// TIA Portal project "e215001v046" (V15)

(* hardware
DEVICE "Estación PC"  SIMATIC PC station
   slot 0: "Estación PC"  Rail  SIMATIC PC-Station  V1.0
      slot 125: "Stationmanager"  Station_Manager  V6.0.4
   slot 1: "IE general_1"  IE General  IE_CP  V8.2.0
   slot 2: "HMI_RT_1"  WinCC RT Advanced  6AV2 104-0xxxx-xxxx  15.0.0.0
      slot 33792: "Interfaz host"  Host interface
DEVICE "HMI_1"  KTP400 Basic mono PN
   slot 0: "HMI_1"  KTP400 Basic mono PN  6AV6 647-0AA11-3AX0  12.0.0.0
   slot 1: "HMI_RT_2"  KTP400 Basic mono PN  6AV6 647-0AA11-3AX0  12.0.0.0
   slot 5: "HMI_1.IE_CP_1"  PROFINET Interface  12.0.0.0
      slot 1: "Interfaz PROFINET_1"  PROFINET Interface
         slot 1: "Port_1"  Port
DEVICE "S7-1200 station_2"  S7-1200 Station
   slot 0: "Rack_0"  S7-1200 Rack  Rack  V1.0
   slot 1: "PLC_1"  CPU 1212C DC/DC/Rly  6ES7 212-1HE31-0XB0  V3.0
*)

// ===== PLC "PLC_1"  CPU 1212C DC/DC/Rly =====

VAR_GLOBAL   // PLC tag table "Tabla de variables estándar"
   "iSensIzqPla1" AT %I0.0 : Bool;
   "iSensMedPla1" AT %I0.1 : Bool;
   "iSensDerPla1" AT %I0.2 : Bool;
   "iMaqProdPla1" AT %I0.3 : Bool;
   "iSensIzqPla2" AT %I0.4 : Bool;
   "iSensMedPla2" AT %I0.5 : Bool;
   "iSensDerPla2" AT %I0.6 : Bool;
   "iMaqProdPla2" AT %I0.7 : Bool;
   "System_Byte" AT %MB1 : Byte;
   "FirstScan" AT %M1.0 : Bool;
   "DiagStatusUpdate" AT %M1.1 : Bool;
   "AlwaysTRUE" AT %M1.2 : Bool;
   "AlwaysFALSE" AT %M1.3 : Bool;
   "Clock_Byte" AT %MB0 : Byte;
   "Clock_10Hz" AT %M0.0 : Bool;
   "Clock_5Hz" AT %M0.1 : Bool;
   "Clock_2.5Hz" AT %M0.2 : Bool;
   "Clock_2Hz" AT %M0.3 : Bool;
   "Clock_1.25Hz" AT %M0.4 : Bool;
   "Clock_1Hz" AT %M0.5 : Bool;
   "Clock_0.625Hz" AT %M0.6 : Bool;
   "Clock_0.5Hz" AT %M0.7 : Bool;
   "fClock_10Hz" AT %M2.0 : Bool;
   "xClock_10Hz" AT %M2.1 : Bool;
   "Plan1EnProd" AT %M2.2 : Bool;
   "Plan1Ok" AT %M2.3 : Bool;
   "Tag_1" AT %M10.0 : Bool;
   "Tag_2" AT %M10.1 : Bool;
   "Tag_3" AT %M10.2 : Bool;
   "Tag_4" AT %M10.3 : Bool;
   "Tag_5" AT %M11.0 : Bool;
   "Tag_6" AT %M11.1 : Bool;
   "Tag_7" AT %M11.2 : Bool;
   "Tag_8" AT %M11.3 : Bool;
   "Flc_Asc_Planch1_10Hz" AT %M501.0 : Bool;
   "Flc_Asc_Planch2_10Hz" AT %M501.1 : Bool;
   "Rec_Alarm" AT %M5.0 : Bool;
   "Osc_5mins" AT %M100.0 : Bool;
   "Palabra Distr" AT %MB101 : Byte;
   "PFlc_SnsMed" AT %M100.1 : Bool;
   "Act_Simu" AT %M1000.0 : Bool;
   "HMI_Supervisor_Actual" AT %M50.0 : Bool;
   "periodoPlanchas" AT %MD110 : DInt;
   "promedioAvanceReal" AT %MD114 : Real;
   "contPromAvReal" AT %MD118 : DInt;
   "tmp_avanceReal_1" AT %MD122 : Real;
   "doProm" AT %M50.1 : Bool;
   "doProm_calculo" AT %M50.2 : Bool;
   "promDone" AT %M50.3 : Bool;
   "Tag_9" AT %M50.4 : Bool;
END_VAR

VAR_GLOBAL   // PLC tag table "DIDO"
   "fSup1" AT %M2.4 : Bool;
   "xsup1" AT %M2.5 : Bool;
   "fSup2" AT %M2.6 : Bool;
   "xsup2" AT %M2.7 : Bool;
   "fSup3" AT %M3.0 : Bool;
   "xsup3" AT %M3.1 : Bool;
   "fSup4" AT %M3.2 : Bool;
   "xsup4" AT %M3.3 : Bool;
   "Cada15M" AT %M3.4 : Bool;
   "fCada15M" AT %M3.5 : Bool;
   "xCada15M" AT %M3.6 : Bool;
   "Supervision" AT %M3.7 : Bool;
   "Plan2EnProd" AT %M4.3 : Bool;
   "Plan2Ok" AT %M4.7 : Bool;
END_VAR

DATA_BLOCK "Planchadora1"   // DB1
{ S7_Optimized_Access := 'TRUE' }
VERSION : 0.1
   VAR RETAIN
      Operadores : Array[1..10] of Struct
         Tiempo : DInt;
         Produccion : DInt;
         Productividad : DInt;
         Sensor : DInt;
         Rendimiento : DInt;
         RendPesado : DInt;
         Estado : Bool;
         Diadelasemana : Array[1..7] of Struct
            Entrda : Time_Of_Day;
            Salida : Time_Of_Day;
         END_STRUCT;
      END_STRUCT;
      Supervisores : Array[1..4] of Struct
         Tiempo : DInt;
         Produccion : DInt;
         Productividad : DInt;
         Sensor : DInt;
         Rendimiento : DInt;
         RendPesado : DInt;
         Estado : Bool;
         Diadelasemana : Array[1..7] of Struct
            Entrada : Time_Of_Day;
            Salida : Time_Of_Day;
            CantOp : Int;
         END_STRUCT;
      END_STRUCT;
      FechaHoraPLC : DTL := DTL#2020-03-12-10:25:17.055662;
      ProductividadTotal : DInt := 861_100_900;
      Productividad : DInt := 0;
      Productividad_100 : Real := 0.0;
      TiempoTotal : DInt := 978_227_090;
      Tiempo : DInt := 511710;
      RendimientoTotal : DInt := 246_159_997;
      Rendimiento : DInt := 0;
   END_VAR
   VAR
      DifRendimiento : DInt := 0;
   END_VAR
   VAR RETAIN
      Rendimiento_100 : Real := 39.44824;
      RendPesado : DInt := 244_381_165;
      RendPesado_100 : Real := 970325.3;
      Productividad_Verde : Real := 0.0;
      Productividad_Amarillo : Real := 0.0;
      Productividad_Rojo : Real := 0.0;
      Rendimiento_Verde : Real := 0.0;
      Rendimiento_Amarillo : Real := 0.0;
      Rendimiento_Rojo : Real := 0.0;
      Peso_Sensor : Int := 0;
      Peso_SensorIZq : Int := 0;
      Peso_SensorDer : Int := 0;
      Peso_SensorMed : Int := 0;
      TiempoCada15 : DInt := 0;
      ProductividadCada15 : DInt := 0;
      RendimientoCada15 : DInt := 0;
      TiempoCada15Ant : DInt := 978_165_380;
      ProductividadCada15Ant : DInt := 861_100_900;
      RendimientoCada15Ant : DInt := 246_159_997;
      EstadoSsIzq : Byte := 16#00;
      EstadoSsDer : Byte := 16#00;
      EstadoSSMed : Byte := 16#00;
   END_VAR
   VAR
      SumaOperario : Int := 1;
   END_VAR
   VAR RETAIN
      FactorCorrRend : Real := 2.0;
   END_VAR
BEGIN
   Operadores[1].Tiempo := 0;
   Operadores[1].Produccion := 0;
   Operadores[1].Productividad := 0;
   Operadores[1].Sensor := 0;
   Operadores[1].Rendimiento := 0;
   Operadores[1].RendPesado := 0;
   Operadores[1].Estado := FALSE;
   Operadores[1].Diadelasemana[1].Entrda := TOD#00:00:00;
   Operadores[1].Diadelasemana[1].Salida := TOD#00:00:00;
   Operadores[1].Diadelasemana[2].Entrda := TOD#00:00:00;
   Operadores[1].Diadelasemana[2].Salida := TOD#00:00:00;
   Operadores[1].Diadelasemana[3].Entrda := TOD#00:00:00;
   Operadores[1].Diadelasemana[3].Salida := TOD#00:00:00;
   Operadores[1].Diadelasemana[4].Entrda := TOD#00:00:00;
   Operadores[1].Diadelasemana[4].Salida := TOD#00:00:00;
   Operadores[1].Diadelasemana[5].Entrda := TOD#00:00:00;
   Operadores[1].Diadelasemana[5].Salida := TOD#00:00:00;
   Operadores[1].Diadelasemana[6].Entrda := TOD#00:00:00;
   Operadores[1].Diadelasemana[6].Salida := TOD#00:00:00;
   Operadores[1].Diadelasemana[7].Entrda := TOD#00:00:00;
   Operadores[1].Diadelasemana[7].Salida := TOD#00:00:00;
   Operadores[2].Tiempo := 0;
   Operadores[2].Produccion := 0;
   Operadores[2].Productividad := 0;
   Operadores[2].Sensor := 0;
   Operadores[2].Rendimiento := 0;
   Operadores[2].RendPesado := 0;
   Operadores[2].Estado := FALSE;
   Operadores[2].Diadelasemana[1].Entrda := TOD#00:00:00;
   Operadores[2].Diadelasemana[1].Salida := TOD#00:00:00;
   Operadores[2].Diadelasemana[2].Entrda := TOD#00:00:00;
   Operadores[2].Diadelasemana[2].Salida := TOD#00:00:00;
   Operadores[2].Diadelasemana[3].Entrda := TOD#00:00:00;
   Operadores[2].Diadelasemana[3].Salida := TOD#00:00:00;
   Operadores[2].Diadelasemana[4].Entrda := TOD#00:00:00;
   Operadores[2].Diadelasemana[4].Salida := TOD#00:00:00;
   Operadores[2].Diadelasemana[5].Entrda := TOD#00:00:00;
   Operadores[2].Diadelasemana[5].Salida := TOD#00:00:00;
   Operadores[2].Diadelasemana[6].Entrda := TOD#00:00:00;
   Operadores[2].Diadelasemana[6].Salida := TOD#00:00:00;
   Operadores[2].Diadelasemana[7].Entrda := TOD#00:00:00;
   Operadores[2].Diadelasemana[7].Salida := TOD#00:00:00;
   Operadores[3].Tiempo := 0;
   Operadores[3].Produccion := 0;
   Operadores[3].Productividad := 0;
   Operadores[3].Sensor := 0;
   Operadores[3].Rendimiento := 0;
   Operadores[3].RendPesado := 0;
   Operadores[3].Estado := FALSE;
   Operadores[3].Diadelasemana[1].Entrda := TOD#00:00:00;
   Operadores[3].Diadelasemana[1].Salida := TOD#00:00:00;
   Operadores[3].Diadelasemana[2].Entrda := TOD#00:00:00;
   Operadores[3].Diadelasemana[2].Salida := TOD#00:00:00;
   Operadores[3].Diadelasemana[3].Entrda := TOD#00:00:00;
   Operadores[3].Diadelasemana[3].Salida := TOD#00:00:00;
   Operadores[3].Diadelasemana[4].Entrda := TOD#00:00:00;
   Operadores[3].Diadelasemana[4].Salida := TOD#00:00:00;
   Operadores[3].Diadelasemana[5].Entrda := TOD#00:00:00;
   Operadores[3].Diadelasemana[5].Salida := TOD#00:00:00;
   Operadores[3].Diadelasemana[6].Entrda := TOD#00:00:00;
   Operadores[3].Diadelasemana[6].Salida := TOD#00:00:00;
   Operadores[3].Diadelasemana[7].Entrda := TOD#00:00:00;
   Operadores[3].Diadelasemana[7].Salida := TOD#00:00:00;
   Operadores[4].Tiempo := 55366140;
   Operadores[4].Produccion := 49275400;
   Operadores[4].Productividad := 0;
   Operadores[4].Sensor := 0;
   Operadores[4].Rendimiento := 12680067;
   Operadores[4].RendPesado := 12605331;
   Operadores[4].Estado := FALSE;
   Operadores[4].Diadelasemana[1].Entrda := TOD#00:00:00;
   Operadores[4].Diadelasemana[1].Salida := TOD#00:00:00;
   Operadores[4].Diadelasemana[2].Entrda := TOD#00:00:00;
   Operadores[4].Diadelasemana[2].Salida := TOD#00:00:00;
   Operadores[4].Diadelasemana[3].Entrda := TOD#00:00:00;
   Operadores[4].Diadelasemana[3].Salida := TOD#00:00:00;
   Operadores[4].Diadelasemana[4].Entrda := TOD#00:00:00;
   Operadores[4].Diadelasemana[4].Salida := TOD#00:00:00;
   Operadores[4].Diadelasemana[5].Entrda := TOD#00:00:00;
   Operadores[4].Diadelasemana[5].Salida := TOD#00:00:00;
   Operadores[4].Diadelasemana[6].Entrda := TOD#00:00:00;
   Operadores[4].Diadelasemana[6].Salida := TOD#00:00:00;
   Operadores[4].Diadelasemana[7].Entrda := TOD#00:00:00;
   Operadores[4].Diadelasemana[7].Salida := TOD#00:00:00;
   Operadores[5].Tiempo := 976_354_630;
   Operadores[5].Produccion := 859_251_080;
   Operadores[5].Productividad := 0;
   Operadores[5].Sensor := 0;
   Operadores[5].Rendimiento := 245_655_295;
   Operadores[5].RendPesado := 243_132_090;
   Operadores[5].Estado := TRUE;
   Operadores[5].Diadelasemana[1].Entrda := TOD#00:00:00;
   Operadores[5].Diadelasemana[1].Salida := TOD#00:00:00;
   Operadores[5].Diadelasemana[2].Entrda := TOD#00:00:00;
   Operadores[5].Diadelasemana[2].Salida := TOD#00:00:00;
   Operadores[5].Diadelasemana[3].Entrda := TOD#00:00:00;
   Operadores[5].Diadelasemana[3].Salida := TOD#00:00:00;
   Operadores[5].Diadelasemana[4].Entrda := TOD#00:00:00;
   Operadores[5].Diadelasemana[4].Salida := TOD#00:00:00;
   Operadores[5].Diadelasemana[5].Entrda := TOD#00:00:00;
   Operadores[5].Diadelasemana[5].Salida := TOD#00:00:00;
   Operadores[5].Diadelasemana[6].Entrda := TOD#00:00:00;
   Operadores[5].Diadelasemana[6].Salida := TOD#00:00:00;
   Operadores[5].Diadelasemana[7].Entrda := TOD#00:00:00;
   Operadores[5].Diadelasemana[7].Salida := TOD#00:00:00;
   Operadores[6].Tiempo := 0;
   Operadores[6].Produccion := 0;
   Operadores[6].Productividad := 0;
   Operadores[6].Sensor := 0;
   Operadores[6].Rendimiento := 0;
   Operadores[6].RendPesado := 0;
   Operadores[6].Estado := FALSE;
   Operadores[6].Diadelasemana[1].Entrda := TOD#00:00:00;
   Operadores[6].Diadelasemana[1].Salida := TOD#00:00:00;
   Operadores[6].Diadelasemana[2].Entrda := TOD#00:00:00;
   Operadores[6].Diadelasemana[2].Salida := TOD#00:00:00;
   Operadores[6].Diadelasemana[3].Entrda := TOD#00:00:00;
   Operadores[6].Diadelasemana[3].Salida := TOD#00:00:00;
   Operadores[6].Diadelasemana[4].Entrda := TOD#00:00:00;
   Operadores[6].Diadelasemana[4].Salida := TOD#00:00:00;
   Operadores[6].Diadelasemana[5].Entrda := TOD#00:00:00;
   Operadores[6].Diadelasemana[5].Salida := TOD#00:00:00;
   Operadores[6].Diadelasemana[6].Entrda := TOD#00:00:00;
   Operadores[6].Diadelasemana[6].Salida := TOD#00:00:00;
   Operadores[6].Diadelasemana[7].Entrda := TOD#00:00:00;
   Operadores[6].Diadelasemana[7].Salida := TOD#00:00:00;
   Operadores[7].Tiempo := 0;
   Operadores[7].Produccion := 0;
   Operadores[7].Productividad := 0;
   Operadores[7].Sensor := 0;
   Operadores[7].Rendimiento := 0;
   Operadores[7].RendPesado := 0;
   Operadores[7].Estado := FALSE;
   Operadores[7].Diadelasemana[1].Entrda := TOD#00:00:00;
   Operadores[7].Diadelasemana[1].Salida := TOD#00:00:00;
   Operadores[7].Diadelasemana[2].Entrda := TOD#00:00:00;
   Operadores[7].Diadelasemana[2].Salida := TOD#00:00:00;
   Operadores[7].Diadelasemana[3].Entrda := TOD#00:00:00;
   Operadores[7].Diadelasemana[3].Salida := TOD#00:00:00;
   Operadores[7].Diadelasemana[4].Entrda := TOD#00:00:00;
   Operadores[7].Diadelasemana[4].Salida := TOD#00:00:00;
   Operadores[7].Diadelasemana[5].Entrda := TOD#00:00:00;
   Operadores[7].Diadelasemana[5].Salida := TOD#00:00:00;
   Operadores[7].Diadelasemana[6].Entrda := TOD#00:00:00;
   Operadores[7].Diadelasemana[6].Salida := TOD#00:00:00;
   Operadores[7].Diadelasemana[7].Entrda := TOD#00:00:00;
   Operadores[7].Diadelasemana[7].Salida := TOD#00:00:00;
   Operadores[8].Tiempo := 0;
   Operadores[8].Produccion := 0;
   Operadores[8].Productividad := 0;
   Operadores[8].Sensor := 0;
   Operadores[8].Rendimiento := 0;
   Operadores[8].RendPesado := 0;
   Operadores[8].Estado := FALSE;
   Operadores[8].Diadelasemana[1].Entrda := TOD#00:00:00;
   Operadores[8].Diadelasemana[1].Salida := TOD#00:00:00;
   Operadores[8].Diadelasemana[2].Entrda := TOD#00:00:00;
   Operadores[8].Diadelasemana[2].Salida := TOD#00:00:00;
   Operadores[8].Diadelasemana[3].Entrda := TOD#00:00:00;
   Operadores[8].Diadelasemana[3].Salida := TOD#00:00:00;
   Operadores[8].Diadelasemana[4].Entrda := TOD#00:00:00;
   Operadores[8].Diadelasemana[4].Salida := TOD#00:00:00;
   Operadores[8].Diadelasemana[5].Entrda := TOD#00:00:00;
   Operadores[8].Diadelasemana[5].Salida := TOD#00:00:00;
   Operadores[8].Diadelasemana[6].Entrda := TOD#00:00:00;
   Operadores[8].Diadelasemana[6].Salida := TOD#00:00:00;
   Operadores[8].Diadelasemana[7].Entrda := TOD#00:00:00;
   Operadores[8].Diadelasemana[7].Salida := TOD#00:00:00;
   Operadores[9].Tiempo := 0;
   Operadores[9].Produccion := 0;
   Operadores[9].Productividad := 0;
   Operadores[9].Sensor := 0;
   Operadores[9].Rendimiento := 0;
   Operadores[9].RendPesado := 0;
   Operadores[9].Estado := FALSE;
   Operadores[9].Diadelasemana[1].Entrda := TOD#00:00:00;
   Operadores[9].Diadelasemana[1].Salida := TOD#00:00:00;
   Operadores[9].Diadelasemana[2].Entrda := TOD#00:00:00;
   Operadores[9].Diadelasemana[2].Salida := TOD#00:00:00;
   Operadores[9].Diadelasemana[3].Entrda := TOD#00:00:00;
   Operadores[9].Diadelasemana[3].Salida := TOD#00:00:00;
   Operadores[9].Diadelasemana[4].Entrda := TOD#00:00:00;
   Operadores[9].Diadelasemana[4].Salida := TOD#00:00:00;
   Operadores[9].Diadelasemana[5].Entrda := TOD#00:00:00;
   Operadores[9].Diadelasemana[5].Salida := TOD#00:00:00;
   Operadores[9].Diadelasemana[6].Entrda := TOD#00:00:00;
   Operadores[9].Diadelasemana[6].Salida := TOD#00:00:00;
   Operadores[9].Diadelasemana[7].Entrda := TOD#00:00:00;
   Operadores[9].Diadelasemana[7].Salida := TOD#00:00:00;
   Operadores[10].Tiempo := 2860;
   Operadores[10].Produccion := 2860;
   Operadores[10].Productividad := 0;
   Operadores[10].Sensor := 0;
   Operadores[10].Rendimiento := 281;
   Operadores[10].RendPesado := 0;
   Operadores[10].Estado := FALSE;
   Operadores[10].Diadelasemana[1].Entrda := TOD#00:00:00;
   Operadores[10].Diadelasemana[1].Salida := TOD#00:00:00;
   Operadores[10].Diadelasemana[2].Entrda := TOD#00:00:00;
   Operadores[10].Diadelasemana[2].Salida := TOD#00:00:00;
   Operadores[10].Diadelasemana[3].Entrda := TOD#00:00:00;
   Operadores[10].Diadelasemana[3].Salida := TOD#00:00:00;
   Operadores[10].Diadelasemana[4].Entrda := TOD#00:00:00;
   Operadores[10].Diadelasemana[4].Salida := TOD#00:00:00;
   Operadores[10].Diadelasemana[5].Entrda := TOD#00:00:00;
   Operadores[10].Diadelasemana[5].Salida := TOD#00:00:00;
   Operadores[10].Diadelasemana[6].Entrda := TOD#00:00:00;
   Operadores[10].Diadelasemana[6].Salida := TOD#00:00:00;
   Operadores[10].Diadelasemana[7].Entrda := TOD#00:00:00;
   Operadores[10].Diadelasemana[7].Salida := TOD#00:00:00;
   Supervisores[1].Tiempo := 253_394_970;
   Supervisores[1].Produccion := 229_902_840;
   Supervisores[1].Productividad := 0;
   Supervisores[1].Sensor := 0;
   Supervisores[1].Rendimiento := 65119768;
   Supervisores[1].RendPesado := 2880135;
   Supervisores[1].Estado := FALSE;
   Supervisores[1].Diadelasemana[1].Entrada := TOD#00:00:00;
   Supervisores[1].Diadelasemana[1].Salida := TOD#00:00:00;
   Supervisores[1].Diadelasemana[1].CantOp := 1;
   Supervisores[1].Diadelasemana[2].Entrada := TOD#06:00:00;
   Supervisores[1].Diadelasemana[2].Salida := TOD#09:00:00;
   Supervisores[1].Diadelasemana[2].CantOp := 1;
   Supervisores[1].Diadelasemana[3].Entrada := TOD#06:00:00;
   Supervisores[1].Diadelasemana[3].Salida := TOD#09:00:00;
   Supervisores[1].Diadelasemana[3].CantOp := 1;
   Supervisores[1].Diadelasemana[4].Entrada := TOD#06:00:00;
   Supervisores[1].Diadelasemana[4].Salida := TOD#09:00:00;
   Supervisores[1].Diadelasemana[4].CantOp := 1;
   Supervisores[1].Diadelasemana[5].Entrada := TOD#06:00:00;
   Supervisores[1].Diadelasemana[5].Salida := TOD#09:00:00;
   Supervisores[1].Diadelasemana[5].CantOp := 1;
   Supervisores[1].Diadelasemana[6].Entrada := TOD#06:00:00;
   Supervisores[1].Diadelasemana[6].Salida := TOD#09:00:00;
   Supervisores[1].Diadelasemana[6].CantOp := 1;
   Supervisores[1].Diadelasemana[7].Entrada := TOD#06:00:00;
   Supervisores[1].Diadelasemana[7].Salida := TOD#14:00:00;
   Supervisores[1].Diadelasemana[7].CantOp := 1;
   Supervisores[2].Tiempo := 427_440_520;
   Supervisores[2].Produccion := 385_662_930;
   Supervisores[2].Productividad := 0;
   Supervisores[2].Sensor := 0;
   Supervisores[2].Rendimiento := 113_827_501;
   Supervisores[2].RendPesado := 3250056;
   Supervisores[2].Estado := TRUE;
   Supervisores[2].Diadelasemana[1].Entrada := TOD#00:00:00;
   Supervisores[2].Diadelasemana[1].Salida := TOD#00:00:00;
   Supervisores[2].Diadelasemana[1].CantOp := 1;
   Supervisores[2].Diadelasemana[2].Entrada := TOD#09:00:00;
   Supervisores[2].Diadelasemana[2].Salida := TOD#17:00:00;
   Supervisores[2].Diadelasemana[2].CantOp := 1;
   Supervisores[2].Diadelasemana[3].Entrada := TOD#09:00:00;
   Supervisores[2].Diadelasemana[3].Salida := TOD#17:00:00;
   Supervisores[2].Diadelasemana[3].CantOp := 1;
   Supervisores[2].Diadelasemana[4].Entrada := TOD#09:00:00;
   Supervisores[2].Diadelasemana[4].Salida := TOD#17:00:00;
   Supervisores[2].Diadelasemana[4].CantOp := 1;
   Supervisores[2].Diadelasemana[5].Entrada := TOD#09:00:00;
   Supervisores[2].Diadelasemana[5].Salida := TOD#17:00:00;
   Supervisores[2].Diadelasemana[5].CantOp := 1;
   Supervisores[2].Diadelasemana[6].Entrada := TOD#09:00:00;
   Supervisores[2].Diadelasemana[6].Salida := TOD#17:00:00;
   Supervisores[2].Diadelasemana[6].CantOp := 1;
   Supervisores[2].Diadelasemana[7].Entrada := TOD#14:00:00;
   Supervisores[2].Diadelasemana[7].Salida := TOD#22:00:00;
   Supervisores[2].Diadelasemana[7].CantOp := 1;
   Supervisores[3].Tiempo := 297_391_250;
   Supervisores[3].Produccion := 245_534_940;
   Supervisores[3].Productividad := 0;
   Supervisores[3].Sensor := 0;
   Supervisores[3].Rendimiento := 67212726;
   Supervisores[3].RendPesado := 2469772;
   Supervisores[3].Estado := FALSE;
   Supervisores[3].Diadelasemana[1].Entrada := TOD#06:00:00;
   Supervisores[3].Diadelasemana[1].Salida := TOD#14:00:00;
   Supervisores[3].Diadelasemana[1].CantOp := 1;
   Supervisores[3].Diadelasemana[2].Entrada := TOD#17:00:00;
   Supervisores[3].Diadelasemana[2].Salida := TOD#22:00:00;
   Supervisores[3].Diadelasemana[2].CantOp := 1;
   Supervisores[3].Diadelasemana[3].Entrada := TOD#17:00:00;
   Supervisores[3].Diadelasemana[3].Salida := TOD#22:00:00;
   Supervisores[3].Diadelasemana[3].CantOp := 1;
   Supervisores[3].Diadelasemana[4].Entrada := TOD#17:00:00;
   Supervisores[3].Diadelasemana[4].Salida := TOD#22:00:00;
   Supervisores[3].Diadelasemana[4].CantOp := 1;
   Supervisores[3].Diadelasemana[5].Entrada := TOD#17:00:00;
   Supervisores[3].Diadelasemana[5].Salida := TOD#22:00:00;
   Supervisores[3].Diadelasemana[5].CantOp := 1;
   Supervisores[3].Diadelasemana[6].Entrada := TOD#17:00:00;
   Supervisores[3].Diadelasemana[6].Salida := TOD#22:00:00;
   Supervisores[3].Diadelasemana[6].CantOp := 1;
   Supervisores[3].Diadelasemana[7].Entrada := TOD#00:00:00;
   Supervisores[3].Diadelasemana[7].Salida := TOD#00:00:00;
   Supervisores[3].Diadelasemana[7].CantOp := 1;
   Supervisores[4].Tiempo := 0;
   Supervisores[4].Produccion := 0;
   Supervisores[4].Productividad := 0;
   Supervisores[4].Sensor := 0;
   Supervisores[4].Rendimiento := 0;
   Supervisores[4].RendPesado := 0;
   Supervisores[4].Estado := FALSE;
   Supervisores[4].Diadelasemana[1].Entrada := TOD#00:00:00;
   Supervisores[4].Diadelasemana[1].Salida := TOD#00:00:00;
   Supervisores[4].Diadelasemana[1].CantOp := 1;
   Supervisores[4].Diadelasemana[2].Entrada := TOD#00:00:00;
   Supervisores[4].Diadelasemana[2].Salida := TOD#00:00:00;
   Supervisores[4].Diadelasemana[2].CantOp := 1;
   Supervisores[4].Diadelasemana[3].Entrada := TOD#00:00:00;
   Supervisores[4].Diadelasemana[3].Salida := TOD#00:00:00;
   Supervisores[4].Diadelasemana[3].CantOp := 1;
   Supervisores[4].Diadelasemana[4].Entrada := TOD#00:00:00;
   Supervisores[4].Diadelasemana[4].Salida := TOD#00:00:00;
   Supervisores[4].Diadelasemana[4].CantOp := 1;
   Supervisores[4].Diadelasemana[5].Entrada := TOD#00:00:00;
   Supervisores[4].Diadelasemana[5].Salida := TOD#00:00:00;
   Supervisores[4].Diadelasemana[5].CantOp := 1;
   Supervisores[4].Diadelasemana[6].Entrada := TOD#00:00:00;
   Supervisores[4].Diadelasemana[6].Salida := TOD#00:00:00;
   Supervisores[4].Diadelasemana[6].CantOp := 1;
   Supervisores[4].Diadelasemana[7].Entrada := TOD#00:00:00;
   Supervisores[4].Diadelasemana[7].Salida := TOD#00:00:00;
   Supervisores[4].Diadelasemana[7].CantOp := 1;
END_DATA_BLOCK

DATA_BLOCK "Planchadora2"   // DB5
{ S7_Optimized_Access := 'TRUE' }
VERSION : 0.1
   VAR RETAIN
      Operadores : Array[1..10] of Struct
         Tiempo : DInt;
         Produccion : DInt;
         Productividad : DInt;
         Sensor : DInt;
         Rendimiento : DInt;
         RendPesado : DInt;
         Estado : Bool;
         Diadelasemana : Array[1..7] of Struct
            Entrda : Time_Of_Day;
            Salida : Time_Of_Day;
         END_STRUCT;
      END_STRUCT;
      Supervisores : Array[1..4] of Struct
         Tiempo : DInt;
         Produccion : DInt;
         Productividad : DInt;
         Sensor : DInt;
         Rendimiento : DInt;
         RendPesado : DInt;
         Estado : Bool;
         Diadelasemana : Array[1..7] of Struct
            Entrada : Time_Of_Day;
            Salida : Time_Of_Day;
            CantOp : Int;
         END_STRUCT;
      END_STRUCT;
      FechaHoraPLC : DTL;
      ProductividadTotal : DInt;
      Productividad : DInt;
      Productividad_100 : Real;
      TiempoTotal : DInt;
      Tiempo : DInt;
      RendimientoTotal : DInt;
      Rendimiento : DInt;
   END_VAR
   VAR
      DifRendimiento : DInt;
   END_VAR
   VAR RETAIN
      Rendimiento_100 : Real;
      RendPesado : DInt;
      RendPesado_100 : Real;
      Productividad_Verde : Real;
      Productividad_Amarillo : Real;
      Productividad_Rojo : Real;
      Rendimiento_Verde : Real;
      Rendimiento_Amarillo : Real;
      Rendimiento_Rojo : Real;
      Peso_Sensor : Int;
      Peso_SensorIZq : Int;
      Peso_SensorDer : Int;
      Peso_SensorMed : Int;
      TiempoCada15 : DInt;
      ProductividadCada15 : DInt;
      RendimientoCada15 : DInt;
      TiempoCada15Ant : DInt;
      ProductividadCada15Ant : DInt;
      RendimientoCada15Ant : DInt;
      EstadoSsIzq : Byte;
      EstadoSsDer : Byte;
      EstadoSSMed : Byte;
      FechayhoraS : String := '1970-01-00-00-00:00:00';
   END_VAR
   VAR
      SumaOperario : Int;
   END_VAR
   VAR RETAIN
      FactorCorrRend : Real := 3.0;
   END_VAR
BEGIN
END_DATA_BLOCK

DATA_BLOCK "Alarmas"   // DB9
{ S7_Optimized_Access := 'FALSE' }
VERSION : 0.1
   VAR
      "PL1-Fall-SnsIzq" : Bool;
      "PL1-Fall-SnsMed" : Bool;
      "PL1-Fall-SnsDer" : Bool;
      "PL2-Fall-SnsIzq" : Bool;
      "PL2-Fall-SnsMed" : Bool;
      "PL2-Fall-SnsDer" : Bool;
      Gen_6 : Bool;
      Gen_7 : Bool;
      Gen_8 : Bool;
      Gen_9 : Bool;
      Gen_10 : Bool;
      Gen_11 : Bool;
      Gen_12 : Bool;
      Gen_13 : Bool;
      Gen_14 : Bool;
      Gen_15 : Bool;
      Gen_16 : Bool;
      Gen_17 : Bool;
      Gen_18 : Bool;
      Gen_19 : Bool;
      Gen_20 : Bool;
      Gen_21 : Bool;
      Gen_22 : Bool;
      Gen_23 : Bool;
      Gen_24 : Bool;
      Gen_25 : Bool;
      Gen_26 : Bool;
      Gen_27 : Bool;
      Gen_28 : Bool;
      Gen_29 : Bool;
      Gen_30 : Bool;
      Gen_31 : Bool;
   END_VAR
BEGIN
END_DATA_BLOCK

DATA_BLOCK "00_ValoresdeReferencia"   // DB11
{ S7_Optimized_Access := 'TRUE' }
VERSION : 0.1
   VAR RETAIN
      pl1_ProdTotal_Ant : DInt;
      pl1_RendTotal_Ant : DInt;
      pl2_ProdTotal_Ant : DInt;
      pl2_RendTotal_Ant : DInt;
   END_VAR
BEGIN
END_DATA_BLOCK

DATA_BLOCK "TratCentecimasSeg"   // DB13
{ S7_Optimized_Access := 'TRUE' }
VERSION : 0.1
   VAR
      Pl1_Cen_SnsIzq : Int;
      Pl1_Cen_SnsMed : Int;
      Pl1_Cen_SnsDer : Int;
      Pl2_Cen_SnsIzq : Int;
      Pl2_Cen_SnsMed : Int;
      Pl2_Cen_SnsDer : Int;
   END_VAR
BEGIN
END_DATA_BLOCK

DATA_BLOCK "Indices"   // DB14
{ S7_Optimized_Access := 'TRUE' }
VERSION : 0.1
   VAR RETAIN
      horasTurno : Time_Of_Day;
      objetivo_100 : Real;
      objetivo : Time_Of_Day;
      avance : Time_Of_Day;
      avance_100 : Real;
      avance_real : Time_Of_Day;
      avance_real_100 : Real;
   END_VAR
BEGIN
END_DATA_BLOCK

// folder: System blocks/Program resources

DATA_BLOCK "tFaSsIzqPl1"   // DB2
{ S7_Optimized_Access := 'TRUE' }
AUTHOR : Simatic
FAMILY : IEC
NAME : IEC_TMR
VERSION : 1.0
// stored: InstanceOfName IEC_TIMER
"IEC_TIMER"
BEGIN
END_DATA_BLOCK

DATA_BLOCK "tFaSsMedPl1"   // DB3
{ S7_Optimized_Access := 'TRUE' }
AUTHOR : Simatic
FAMILY : IEC
NAME : IEC_TMR
VERSION : 1.0
// stored: InstanceOfName IEC_TIMER
"IEC_TIMER"
BEGIN
END_DATA_BLOCK

DATA_BLOCK "tFaSsDerPl1"   // DB4
{ S7_Optimized_Access := 'TRUE' }
AUTHOR : Simatic
FAMILY : IEC
NAME : IEC_TMR
VERSION : 1.0
// stored: InstanceOfName IEC_TIMER
"IEC_TIMER"
BEGIN
END_DATA_BLOCK

DATA_BLOCK "tFaSsIzqPl2"   // DB6
{ S7_Optimized_Access := 'TRUE' }
AUTHOR : Simatic
FAMILY : IEC
NAME : IEC_TMR
VERSION : 1.0
// stored: InstanceOfName IEC_TIMER
"IEC_TIMER"
BEGIN
END_DATA_BLOCK

DATA_BLOCK "tFaSsMedPl2"   // DB7
{ S7_Optimized_Access := 'TRUE' }
AUTHOR : Simatic
FAMILY : IEC
NAME : IEC_TMR
VERSION : 1.0
// stored: InstanceOfName IEC_TIMER
"IEC_TIMER"
BEGIN
END_DATA_BLOCK

DATA_BLOCK "tFaSsDerPl2"   // DB8
{ S7_Optimized_Access := 'TRUE' }
AUTHOR : Simatic
FAMILY : IEC
NAME : IEC_TMR
VERSION : 1.0
// stored: InstanceOfName IEC_TIMER
"IEC_TIMER"
BEGIN
END_DATA_BLOCK

DATA_BLOCK "IEC_Timer_0_DB"   // DB10
{ S7_Optimized_Access := 'TRUE' }
AUTHOR : Simatic
FAMILY : IEC
NAME : IEC_TMR
VERSION : 1.0
// stored: InstanceOfName IEC_TIMER
"IEC_TIMER"
BEGIN
END_DATA_BLOCK

DATA_BLOCK "T_FueradProd"   // DB12
{ S7_Optimized_Access := 'TRUE' }
AUTHOR : Simatic
FAMILY : IEC
NAME : IEC_TMR
VERSION : 1.0
// stored: InstanceOfName IEC_TIMER
"IEC_TIMER"
BEGIN
END_DATA_BLOCK

// folder: (top level)

FUNCTION "GenDatosBD" : Void   // FC1, SCL
{ S7_Optimized_Access := 'TRUE' }
VERSION : 0.1
   VAR_TEMP
      resultado : Int;
      Contador : Int;
      HoraPLC : Time_Of_Day;
      MinutoPLC : USInt;
      HoraSupervisorEntrada : Time_Of_Day;
      HoraSupervisorSalida : Time_Of_Day;
      tmp_HaySupervisor : Bool;
      tmp_StContadorAnt2 : Int;
      tmp_StContadorAnt1 : Int;
      tmp_horaInicio : Time_Of_Day;
      tmp_horaFin : Time_Of_Day;
      tmp_objetivo : Real;
      tmp_avance : DInt;
      tmp_DifRend : DInt;
      tmp_difHora : Time_Of_Day;
      tmp_avance_real_100 : Real;
   END_VAR
BEGIN
   //Leemos el reloj del sistem
   //a y lo guardamos en el DB
   #resultado := RD_LOC_T("Planchadora1".FechaHoraPLC);
   #HoraPLC := DTL_TO_TOD("Planchadora1".FechaHoraPLC);

   #resultado := RD_LOC_T("Planchadora2".FechaHoraPLC);
   #HoraPLC := DTL_TO_TOD("Planchadora2".FechaHoraPLC);

   FOR #Contador := 1 TO 4 DO
       IF "Planchadora1".Supervisores[#Contador].Estado = true THEN
           #tmp_StContadorAnt1 := #Contador;
           #tmp_StContadorAnt2 := #Contador;
       END_IF;
   END_FOR;

   FOR #Contador := 1 TO 4 DO
       //Obtenemos las horas y minutos 
       #HoraSupervisorEntrada := "Planchadora1".Supervisores[#Contador].Diadelasemana["Planchadora1".FechaHoraPLC.WEEKDAY].Entrada;
       #HoraSupervisorSalida  := "Planchadora1".Supervisores[#Contador].Diadelasemana["Planchadora1".FechaHoraPLC.WEEKDAY].Salida;

       //Encendemos o apagamos el Supervisor en función de si la hora está dentro de los valores admitidos
       IF (#HoraPLC >= #HoraSupervisorEntrada) AND (#HoraPLC < #HoraSupervisorSalida) THEN
           #tmp_horaInicio := #HoraSupervisorEntrada;
           #tmp_horaFin := #HoraSupervisorSalida;

           "Planchadora1".Supervisores[#Contador].Estado := true;
           "Planchadora2".Supervisores[#Contador].Estado := true;
           #tmp_HaySupervisor := True;

           // #### CANT DE OPERARIOS SETEADOS DESDE PLANILLA DE HORARIOS
          "Planchadora2".SumaOperario := "Planchadora1".SumaOperario;
           //#######################################################

           IF "fClock_10Hz" THEN
               "Planchadora1".Supervisores[#Contador].Tiempo := "Planchadora1".Supervisores[#Contador].Tiempo + 10;
               IF "Plan1EnProd" THEN
                   "Planchadora1".Supervisores[#Contador].Produccion := "Planchadora1".Supervisores[#Contador].Produccion + 10;
                   "Planchadora1".Supervisores[#Contador].Rendimiento := "Planchadora1".Supervisores[#Contador].Rendimiento + "Planchadora1".Peso_Sensor;
               END_IF;
           END_IF;

           IF "fCada15M" THEN

               IF #tmp_StContadorAnt1 = #Contador THEN
                   "Planchadora1".Supervisores[#Contador].RendPesado := "Planchadora1".Supervisores[#Contador].RendPesado + "Planchadora1".DifRendimiento / "Planchadora1".SumaOperario;
               ELSE
                   "Planchadora1".Supervisores[#tmp_StContadorAnt1].RendPesado := "Planchadora1".Supervisores[#tmp_StContadorAnt1].RendPesado + "Planchadora1".DifRendimiento / "Planchadora1".SumaOperario;
               END_IF;


           END_IF;

           IF "fClock_10Hz" THEN
               "Planchadora2".Supervisores[#Contador].Tiempo := "Planchadora2".Supervisores[#Contador].Tiempo + 10;
               IF "Plan2EnProd" THEN
                   "Planchadora2".Supervisores[#Contador].Produccion := "Planchadora2".Supervisores[#Contador].Produccion + 10;
                   "Planchadora2".Supervisores[#Contador].Rendimiento := "Planchadora2".Supervisores[#Contador].Rendimiento + "Planchadora2".Peso_Sensor;
                  END_IF;
           END_IF;

           IF "fCada15M" THEN
               IF #tmp_StContadorAnt2 = #Contador THEN
                   "Planchadora2".Supervisores[#Contador].RendPesado := "Planchadora2".Supervisores[#Contador].RendPesado + "Planchadora2".DifRendimiento / "Planchadora2".SumaOperario;
               ELSE
                   "Planchadora2".Supervisores[#tmp_StContadorAnt2].RendPesado := "Planchadora2".Supervisores[#tmp_StContadorAnt2].RendPesado + "Planchadora2".DifRendimiento / "Planchadora2".SumaOperario;
               END_IF;
           END_IF;

       ELSE
           "Planchadora1".Supervisores[#Contador].Estado := false;
           "Planchadora2".Supervisores[#Contador].Estado := false;

       END_IF;

   END_FOR;

   IF (#tmp_HaySupervisor = FALSE) THEN
       // Statement section IF
       "Planchadora1".SumaOperario := 0;
       "Planchadora2".SumaOperario := 0;
       ;
   ELSE
       #tmp_HaySupervisor := FALSE;
   END_IF;


   FOR #Contador := 1 TO 10 DO

       IF  "Planchadora1".Operadores[#Contador].Estado THEN
           IF "fClock_10Hz" AND"Supervision" THEN
               "Planchadora1".Operadores[#Contador].Tiempo := "Planchadora1".Operadores[#Contador].Tiempo + 10;
               IF "Plan1EnProd" THEN
                   "Planchadora1".Operadores[#Contador].Produccion := "Planchadora1".Operadores[#Contador].Produccion + 10;
                   "Planchadora1".Operadores[#Contador].Rendimiento := "Planchadora1".Operadores[#Contador].Rendimiento + "Planchadora1".Peso_Sensor;
               END_IF;
           END_IF;

           IF "fCada15M" AND "Supervision" THEN
               "Planchadora1".Operadores[#Contador].RendPesado := "Planchadora1".Operadores[#Contador].RendPesado + "Planchadora1".DifRendimiento / "Planchadora1".SumaOperario;
               // + "Planchadora1".DifRendimiento / "Planchadora1".SumaOperario;
           END_IF;

       END_IF;

       IF "Planchadora2".Operadores[#Contador].Estado THEN
           IF "fClock_10Hz" AND "Plan2Ok" AND "Supervision" THEN
               "Planchadora2".Operadores[#Contador].Tiempo := "Planchadora2".Operadores[#Contador].Tiempo + 10
               ;
               IF "Plan2EnProd" THEN
                   "Planchadora2".Operadores[#Contador].Produccion := "Planchadora2".Operadores[#Contador].Produccion + 10;
                   "Planchadora2".Operadores[#Contador].Rendimiento := "Planchadora2".Operadores[#Contador].Rendimiento + "Planchadora2".Peso_Sensor;
               END_IF;
           END_IF;

           IF "fCada15M" AND "Plan2Ok" AND "Supervision" THEN
               "Planchadora2".Operadores[#Contador].RendPesado := "Planchadora2".Operadores[#Contador].RendPesado + "Planchadora2".DifRendimiento / "Planchadora2".SumaOperario;
           END_IF;

       END_IF;
   END_FOR;

   IF "fCada15M" THEN
       "Planchadora1".RendPesado := "Planchadora1".RendPesado + "Planchadora1".DifRendimiento / "Planchadora1".SumaOperario;
   END_IF;

   IF "fCada15M" AND "Plan2Ok" THEN
       "Planchadora2".RendPesado := "Planchadora2".RendPesado + "Planchadora2".DifRendimiento / "Planchadora2".SumaOperario;
   END_IF;




   #tmp_difHora := T_SUB(IN1:=#tmp_horaFin, IN2:=#tmp_horaInicio);
   IF "Indices".objetivo_100 <> 0 THEN
       #tmp_objetivo := TOD_TO_DINT(#tmp_difHora) * 2 * ("Indices".objetivo_100 / 100);
   END_IF;

   "Indices".objetivo := DINT_TO_TOD(REAL_TO_DINT(#tmp_objetivo));

   "Indices".avance := DINT_TO_TOD(("Planchadora1".Rendimiento + "Planchadora2".Rendimiento) * 10); // trabaja en milis y tengo decimas

   #tmp_avance := "Planchadora1".Rendimiento + "Planchadora2".Rendimiento;

   IF "Planchadora1".Tiempo <> 0 AND "Planchadora2".Tiempo <> 0 THEN
       "Indices".avance_100 := 100 * #tmp_avance / ("Planchadora1".Tiempo + "Planchadora2".Tiempo);
   END_IF;

   #tmp_DifRend := (("Planchadora1".RendimientoTotal - "Planchadora1".RendimientoCada15Ant) + ("Planchadora2".RendimientoTotal - "Planchadora2".RendimientoCada15Ant)) * 10;

   "Indices".avance_real := DINT_TO_TOD(#tmp_DifRend);

   IF "doProm_calculo" THEN

       IF #tmp_DifRend <> 0.0 THEN
           "tmp_avanceReal_1" := 10 * (#tmp_DifRend / ("periodoPlanchas"));
       END_IF;


       #tmp_avance_real_100 := "promedioAvanceReal" * "contPromAvReal";

       #tmp_avance_real_100 := #tmp_avance_real_100 + "tmp_avanceReal_1";

       "contPromAvReal" := "contPromAvReal" + 1;

       "promedioAvanceReal" := #tmp_avance_real_100 / "contPromAvReal";

       IF "promedioAvanceReal" > 0 THEN
           IF "promedioAvanceReal" > 99.0 THEN
               "promedioAvanceReal" := 99.0;
               "Indices".avance_real_100 := 99.0;
           ELSE
               "Indices".avance_real_100 := "promedioAvanceReal";
           END_IF;
       ELSE
           "Indices".avance_real_100 := 0.0;
       END_IF;

       "promDone" := TRUE;

   END_IF;


   // RESET DE VARIABLES
   // 
   IF "Planchadora1".Supervisores[4].Estado = FALSE AND "Planchadora1".Supervisores[1].Estado = FALSE AND "Planchadora1".Supervisores[2].Estado = FALSE AND "Planchadora1".Supervisores[3].Estado = FALSE THEN
       "Indices".avance_real_100 := 0.0;
       "promedioAvanceReal" := 0.0;
       "contPromAvReal" := 0;
   END_IF;
END_FUNCTION

FUNCTION "Plancha1" : Void   // FC2, LAD
{ S7_Optimized_Access := 'FALSE' }
VERSION : 0.1
   VAR_TEMP
      rdiff : DInt;
      pdiff : DInt;
      tdiff : DInt;
      Temp_2 : Bool;
      TempRendPes_1 : Real;
      tmp_Productividad_100 : LReal;
      tmp_Rendimiento_100 : LReal;
      tmp_RendPesado_100 : LReal;
      tmp_Productividad : LReal;
      tmp_Tiempo : LReal;
      tmp_Rendimiento : LReal;
      tmp_RendPesado : LReal;
      tmp_factorCorrRend : DInt;
      Pl1_Prod_Aux1 : DInt;
      Pl1_Rend_Aux1 : DInt;
      Pl1_Fact_Aux1 : Real;
      Pl1_Prod_Aux1_Real : Real;
      Pl1_Rend_Aux1_Real : Real;
   END_VAR
   VAR_TEMP   // added for the SCL form of the ladder/FBD networks
      _w1 : Bool;
      _w2 : Bool;
   END_VAR
BEGIN

REGION Network 1: Inversión de Señal de Sensores
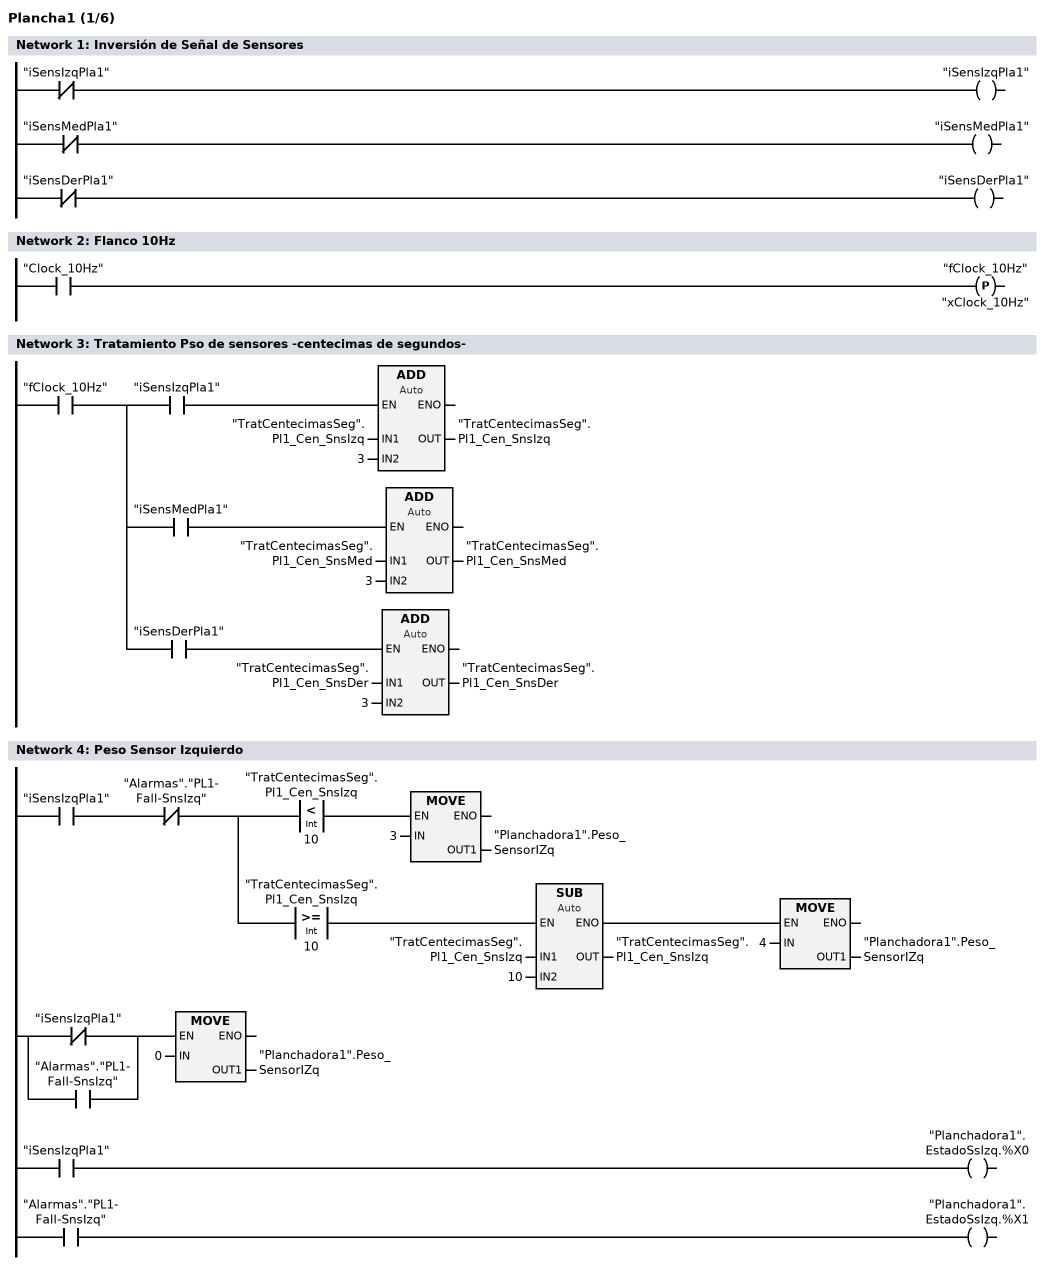
   RUNG wire#powerrail
      I_Contact( "iSensIzqPla1" )
      Coil( "iSensIzqPla1" )
   END_RUNG
   RUNG wire#powerrail
      I_Contact( "iSensMedPla1" )
      Coil( "iSensMedPla1" )
   END_RUNG
   RUNG wire#powerrail
      I_Contact( "iSensDerPla1" )
      Coil( "iSensDerPla1" )
   END_RUNG
   // the same network as SCL:
   "iSensIzqPla1" := NOT "iSensIzqPla1";
   "iSensMedPla1" := NOT "iSensMedPla1";
   "iSensDerPla1" := NOT "iSensDerPla1";
END_REGION

REGION Network 2: Flanco 10Hz
   "fClock_10Hz" := "Clock_10Hz" AND NOT "xClock_10Hz";   // rising edge
   "xClock_10Hz" := "Clock_10Hz";
END_REGION

REGION Network 3: Tratamiento Pso de sensores -centecimas de segundos-
   RUNG wire#powerrail
      Contact( "fClock_10Hz" )
      wire#w1
      Contact( "iSensIzqPla1" )
      { S7_GenerateENO := "TRUE" } Add(in1 := "TratCentecimasSeg".Pl1_Cen_SnsIzq, in2 := 3, out => "TratCentecimasSeg".Pl1_Cen_SnsIzq)
   END_RUNG
   RUNG wire#w1
      Contact( "iSensMedPla1" )
      { S7_GenerateENO := "TRUE" } Add(in1 := "TratCentecimasSeg".Pl1_Cen_SnsMed, in2 := 3, out => "TratCentecimasSeg".Pl1_Cen_SnsMed)
   END_RUNG
   RUNG wire#w1
      Contact( "iSensDerPla1" )
      { S7_GenerateENO := "TRUE" } Add(in1 := "TratCentecimasSeg".Pl1_Cen_SnsDer, in2 := 3, out => "TratCentecimasSeg".Pl1_Cen_SnsDer)
   END_RUNG
   // the same network as SCL:
   IF "fClock_10Hz" AND "iSensIzqPla1" THEN
       "TratCentecimasSeg".Pl1_Cen_SnsIzq := "TratCentecimasSeg".Pl1_Cen_SnsIzq + 3;
   END_IF;
   IF "fClock_10Hz" AND "iSensMedPla1" THEN
       "TratCentecimasSeg".Pl1_Cen_SnsMed := "TratCentecimasSeg".Pl1_Cen_SnsMed + 3;
   END_IF;
   IF "fClock_10Hz" AND "iSensDerPla1" THEN
       "TratCentecimasSeg".Pl1_Cen_SnsDer := "TratCentecimasSeg".Pl1_Cen_SnsDer + 3;
   END_IF;
END_REGION

REGION Network 4: Peso Sensor Izquierdo
   RUNG wire#powerrail
      Contact( "iSensIzqPla1" )
      I_Contact( "Alarmas"."PL1-Fall-SnsIzq" )
      wire#w1
      { S7_Templates := "SrcType := Int" } LT_Contact(in1 := "TratCentecimasSeg".Pl1_Cen_SnsIzq, in2 := 10)
      { S7_GenerateENO := "TRUE" } Move(in := 3, out1 => "Planchadora1".Peso_SensorIZq)
   END_RUNG
   RUNG wire#w1
      { S7_Templates := "SrcType := Int" } GE_Contact(in1 := "TratCentecimasSeg".Pl1_Cen_SnsIzq, in2 := 10)
      { S7_GenerateENO := "TRUE" } Sub(in1 := "TratCentecimasSeg".Pl1_Cen_SnsIzq, in2 := 10, out => "TratCentecimasSeg".Pl1_Cen_SnsIzq)
      { S7_GenerateENO := "TRUE" } Move(in := 4, out1 => "Planchadora1".Peso_SensorIZq)
   END_RUNG
   RUNG wire#powerrail
      I_Contact( "iSensIzqPla1" )
      wire#w2
      { S7_GenerateENO := "TRUE" } Move(in := 0, out1 => "Planchadora1".Peso_SensorIZq)
   END_RUNG
   RUNG wire#powerrail
      Contact( "Alarmas"."PL1-Fall-SnsIzq" )
   END_RUNG wire#w2
   RUNG wire#powerrail
      Contact( "iSensIzqPla1" )
      Coil( "Planchadora1".EstadoSsIzq.%X0 )
   END_RUNG
   RUNG wire#powerrail
      Contact( "Alarmas"."PL1-Fall-SnsIzq" )
      Coil( "Planchadora1".EstadoSsIzq.%X1 )
   END_RUNG
   // the same network as SCL:
   // ENO of a box is taken as its EN; it also drops when the box reports an error
   #_w1 := "iSensIzqPla1" AND NOT "Alarmas"."PL1-Fall-SnsIzq";
   IF #_w1 AND ("TratCentecimasSeg".Pl1_Cen_SnsIzq < 10) THEN "Planchadora1".Peso_SensorIZq := 3; END_IF;
   #_w2 := #_w1 AND ("TratCentecimasSeg".Pl1_Cen_SnsIzq >= 10);
   IF #_w2 THEN
       "TratCentecimasSeg".Pl1_Cen_SnsIzq := "TratCentecimasSeg".Pl1_Cen_SnsIzq - 10;
       "Planchadora1".Peso_SensorIZq := 4;
   END_IF;
   IF NOT "iSensIzqPla1" OR "Alarmas"."PL1-Fall-SnsIzq" THEN "Planchadora1".Peso_SensorIZq := 0; END_IF;
   "Planchadora1".EstadoSsIzq.%X0 := "iSensIzqPla1";
   "Planchadora1".EstadoSsIzq.%X1 := "Alarmas"."PL1-Fall-SnsIzq";
END_REGION

REGION Network 5: Peso Sensor derecho
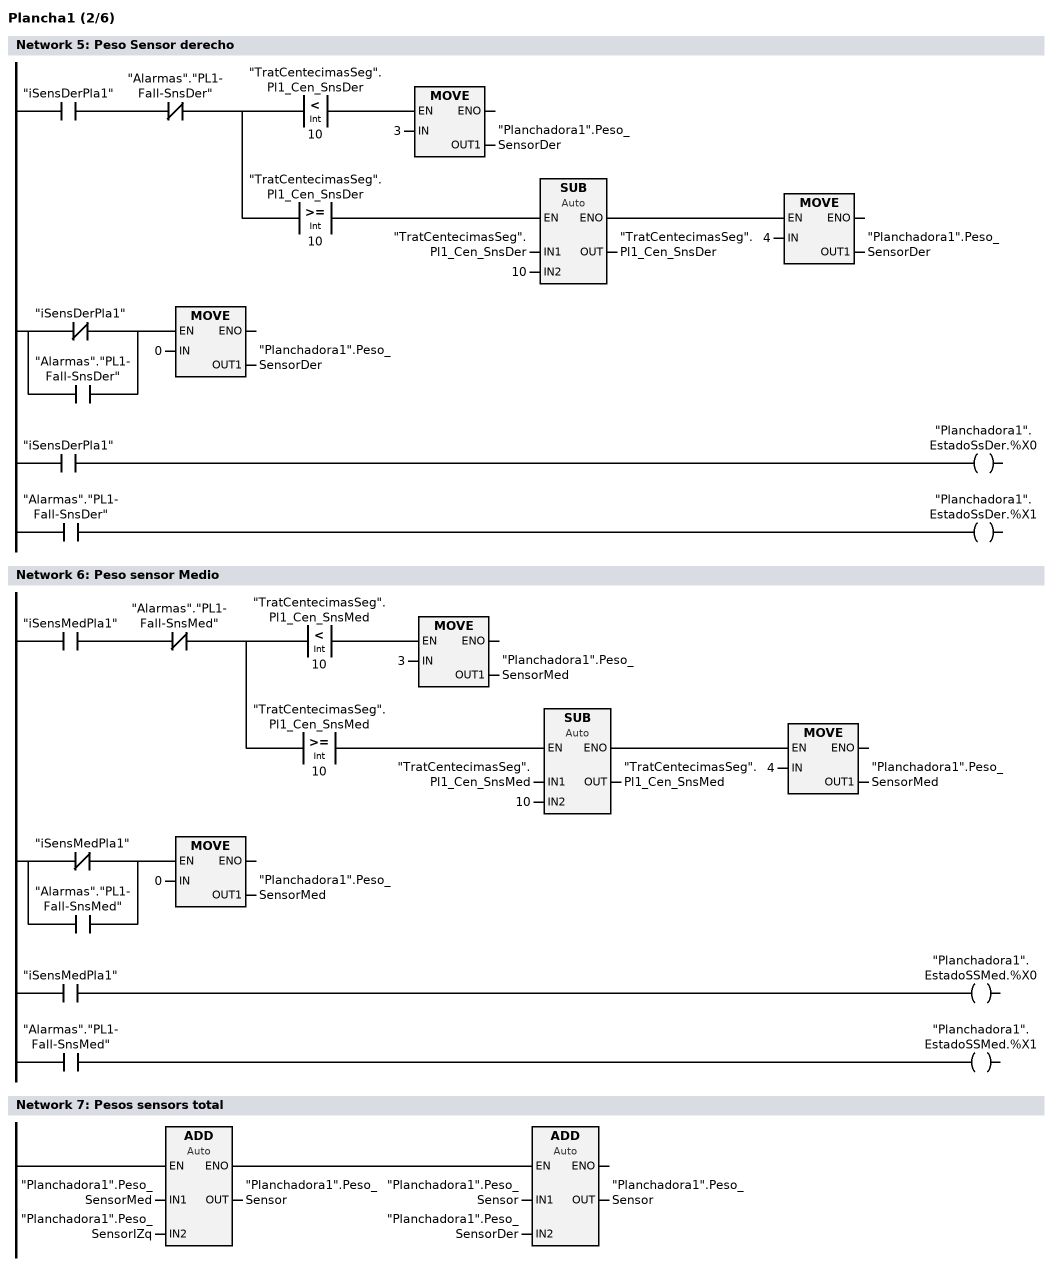
   RUNG wire#powerrail
      Contact( "iSensDerPla1" )
      I_Contact( "Alarmas"."PL1-Fall-SnsDer" )
      wire#w1
      { S7_Templates := "SrcType := Int" } LT_Contact(in1 := "TratCentecimasSeg".Pl1_Cen_SnsDer, in2 := 10)
      { S7_GenerateENO := "TRUE" } Move(in := 3, out1 => "Planchadora1".Peso_SensorDer)
   END_RUNG
   RUNG wire#w1
      { S7_Templates := "SrcType := Int" } GE_Contact(in1 := "TratCentecimasSeg".Pl1_Cen_SnsDer, in2 := 10)
      { S7_GenerateENO := "TRUE" } Sub(in1 := "TratCentecimasSeg".Pl1_Cen_SnsDer, in2 := 10, out => "TratCentecimasSeg".Pl1_Cen_SnsDer)
      { S7_GenerateENO := "TRUE" } Move(in := 4, out1 => "Planchadora1".Peso_SensorDer)
   END_RUNG
   RUNG wire#powerrail
      I_Contact( "iSensDerPla1" )
      wire#w2
      { S7_GenerateENO := "TRUE" } Move(in := 0, out1 => "Planchadora1".Peso_SensorDer)
   END_RUNG
   RUNG wire#powerrail
      Contact( "Alarmas"."PL1-Fall-SnsDer" )
   END_RUNG wire#w2
   RUNG wire#powerrail
      Contact( "iSensDerPla1" )
      Coil( "Planchadora1".EstadoSsDer.%X0 )
   END_RUNG
   RUNG wire#powerrail
      Contact( "Alarmas"."PL1-Fall-SnsDer" )
      Coil( "Planchadora1".EstadoSsDer.%X1 )
   END_RUNG
   // the same network as SCL:
   // ENO of a box is taken as its EN; it also drops when the box reports an error
   #_w1 := "iSensDerPla1" AND NOT "Alarmas"."PL1-Fall-SnsDer";
   IF #_w1 AND ("TratCentecimasSeg".Pl1_Cen_SnsDer < 10) THEN "Planchadora1".Peso_SensorDer := 3; END_IF;
   #_w2 := #_w1 AND ("TratCentecimasSeg".Pl1_Cen_SnsDer >= 10);
   IF #_w2 THEN
       "TratCentecimasSeg".Pl1_Cen_SnsDer := "TratCentecimasSeg".Pl1_Cen_SnsDer - 10;
       "Planchadora1".Peso_SensorDer := 4;
   END_IF;
   IF NOT "iSensDerPla1" OR "Alarmas"."PL1-Fall-SnsDer" THEN "Planchadora1".Peso_SensorDer := 0; END_IF;
   "Planchadora1".EstadoSsDer.%X0 := "iSensDerPla1";
   "Planchadora1".EstadoSsDer.%X1 := "Alarmas"."PL1-Fall-SnsDer";
END_REGION

REGION Network 6: Peso sensor Medio
   RUNG wire#powerrail
      Contact( "iSensMedPla1" )
      I_Contact( "Alarmas"."PL1-Fall-SnsMed" )
      wire#w1
      { S7_Templates := "SrcType := Int" } LT_Contact(in1 := "TratCentecimasSeg".Pl1_Cen_SnsMed, in2 := 10)
      { S7_GenerateENO := "TRUE" } Move(in := 3, out1 => "Planchadora1".Peso_SensorMed)
   END_RUNG
   RUNG wire#w1
      { S7_Templates := "SrcType := Int" } GE_Contact(in1 := "TratCentecimasSeg".Pl1_Cen_SnsMed, in2 := 10)
      { S7_GenerateENO := "TRUE" } Sub(in1 := "TratCentecimasSeg".Pl1_Cen_SnsMed, in2 := 10, out => "TratCentecimasSeg".Pl1_Cen_SnsMed)
      { S7_GenerateENO := "TRUE" } Move(in := 4, out1 => "Planchadora1".Peso_SensorMed)
   END_RUNG
   RUNG wire#powerrail
      I_Contact( "iSensMedPla1" )
      wire#w2
      { S7_GenerateENO := "TRUE" } Move(in := 0, out1 => "Planchadora1".Peso_SensorMed)
   END_RUNG
   RUNG wire#powerrail
      Contact( "Alarmas"."PL1-Fall-SnsMed" )
   END_RUNG wire#w2
   RUNG wire#powerrail
      Contact( "iSensMedPla1" )
      Coil( "Planchadora1".EstadoSSMed.%X0 )
   END_RUNG
   RUNG wire#powerrail
      Contact( "Alarmas"."PL1-Fall-SnsMed" )
      Coil( "Planchadora1".EstadoSSMed.%X1 )
   END_RUNG
   // the same network as SCL:
   // ENO of a box is taken as its EN; it also drops when the box reports an error
   #_w1 := "iSensMedPla1" AND NOT "Alarmas"."PL1-Fall-SnsMed";
   IF #_w1 AND ("TratCentecimasSeg".Pl1_Cen_SnsMed < 10) THEN "Planchadora1".Peso_SensorMed := 3; END_IF;
   #_w2 := #_w1 AND ("TratCentecimasSeg".Pl1_Cen_SnsMed >= 10);
   IF #_w2 THEN
       "TratCentecimasSeg".Pl1_Cen_SnsMed := "TratCentecimasSeg".Pl1_Cen_SnsMed - 10;
       "Planchadora1".Peso_SensorMed := 4;
   END_IF;
   IF NOT "iSensMedPla1" OR "Alarmas"."PL1-Fall-SnsMed" THEN "Planchadora1".Peso_SensorMed := 0; END_IF;
   "Planchadora1".EstadoSSMed.%X0 := "iSensMedPla1";
   "Planchadora1".EstadoSSMed.%X1 := "Alarmas"."PL1-Fall-SnsMed";
END_REGION

REGION Network 7: Pesos sensors total
   RUNG wire#powerrail
      { S7_GenerateENO := "TRUE" } Add(in1 := "Planchadora1".Peso_SensorMed, in2 := "Planchadora1".Peso_SensorIZq, out => "Planchadora1".Peso_Sensor)
      { S7_GenerateENO := "TRUE" } Add(in1 := "Planchadora1".Peso_Sensor, in2 := "Planchadora1".Peso_SensorDer, out => "Planchadora1".Peso_Sensor)
   END_RUNG
   // the same network as SCL:
   // ENO of a box is taken as its EN; it also drops when the box reports an error
   "Planchadora1".Peso_Sensor := "Planchadora1".Peso_SensorMed + "Planchadora1".Peso_SensorIZq;
   "Planchadora1".Peso_Sensor := "Planchadora1".Peso_Sensor + "Planchadora1".Peso_SensorDer;
END_REGION

REGION Network 8: Plancha 1 en produccion
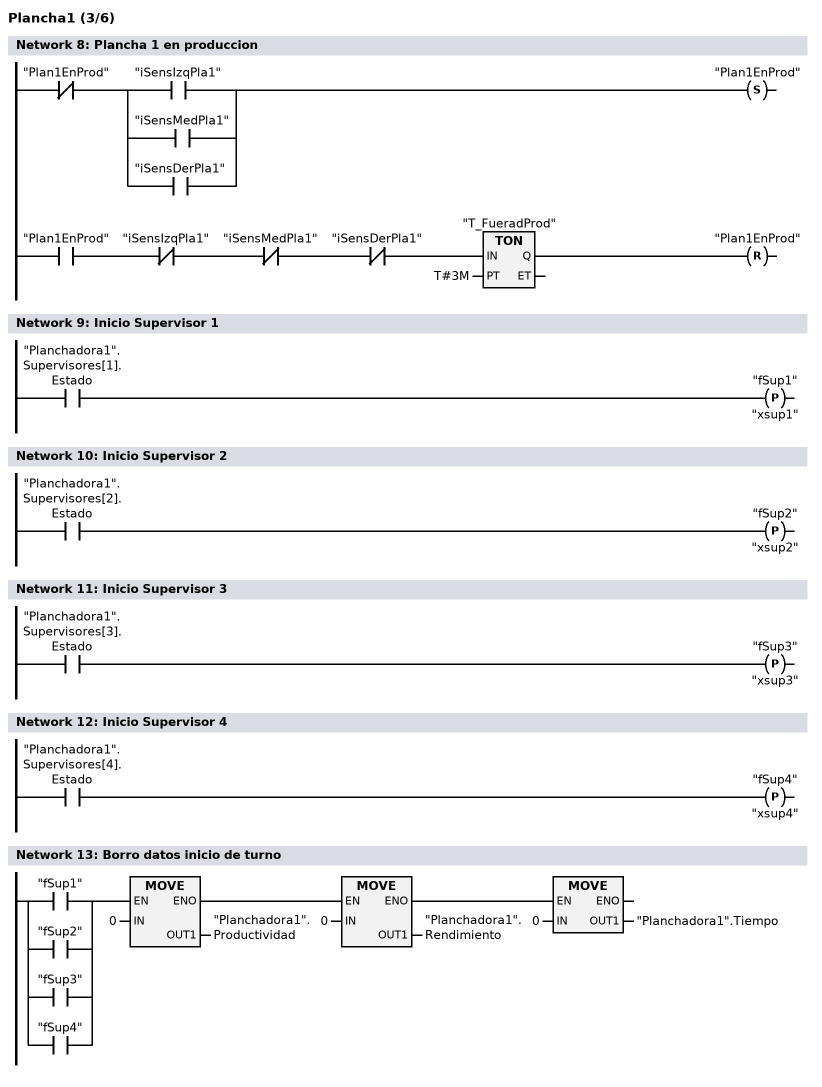
   IF NOT "Plan1EnProd" AND ("iSensIzqPla1" OR "iSensMedPla1" OR "iSensDerPla1") THEN
       "Plan1EnProd" := TRUE;
   END_IF;
   "T_FueradProd".TON(IN := "Plan1EnProd" AND NOT "iSensIzqPla1" AND NOT "iSensMedPla1" AND NOT "iSensDerPla1",
                      PT := T#3M);
   IF "T_FueradProd".Q THEN "Plan1EnProd" := FALSE; END_IF;
END_REGION

REGION Network 9: Inicio Supervisor 1
   "fSup1" := "Planchadora1".Supervisores[1].Estado AND NOT "xsup1";   // rising edge
   "xsup1" := "Planchadora1".Supervisores[1].Estado;
END_REGION

REGION Network 10: Inicio Supervisor 2
   "fSup2" := "Planchadora1".Supervisores[2].Estado AND NOT "xsup2";   // rising edge
   "xsup2" := "Planchadora1".Supervisores[2].Estado;
END_REGION

REGION Network 11: Inicio Supervisor 3
   "fSup3" := "Planchadora1".Supervisores[3].Estado AND NOT "xsup3";   // rising edge
   "xsup3" := "Planchadora1".Supervisores[3].Estado;
END_REGION

REGION Network 12: Inicio Supervisor 4
   "fSup4" := "Planchadora1".Supervisores[4].Estado AND NOT "xsup4";   // rising edge
   "xsup4" := "Planchadora1".Supervisores[4].Estado;
END_REGION

REGION Network 13: Borro datos inicio de turno
   RUNG wire#powerrail
      Contact( "fSup1" )
      wire#w1
      { S7_GenerateENO := "TRUE" } Move(in := 0, out1 => "Planchadora1".Productividad)
      { S7_GenerateENO := "TRUE" } Move(in := 0, out1 => "Planchadora1".Rendimiento)
      { S7_GenerateENO := "TRUE" } Move(in := 0, out1 => "Planchadora1".Tiempo)
   END_RUNG
   RUNG wire#powerrail
      Contact( "fSup2" )
   END_RUNG wire#w1
   RUNG wire#powerrail
      Contact( "fSup3" )
   END_RUNG wire#w1
   RUNG wire#powerrail
      Contact( "fSup4" )
   END_RUNG wire#w1
   // the same network as SCL:
   // ENO of a box is taken as its EN; it also drops when the box reports an error
   IF "fSup1" OR "fSup2" OR "fSup3" OR "fSup4" THEN
       "Planchadora1".Productividad := 0;
       "Planchadora1".Rendimiento := 0;
       "Planchadora1".Tiempo := 0;
   END_IF;
END_REGION

REGION Network 14: Calculo de datos actuales
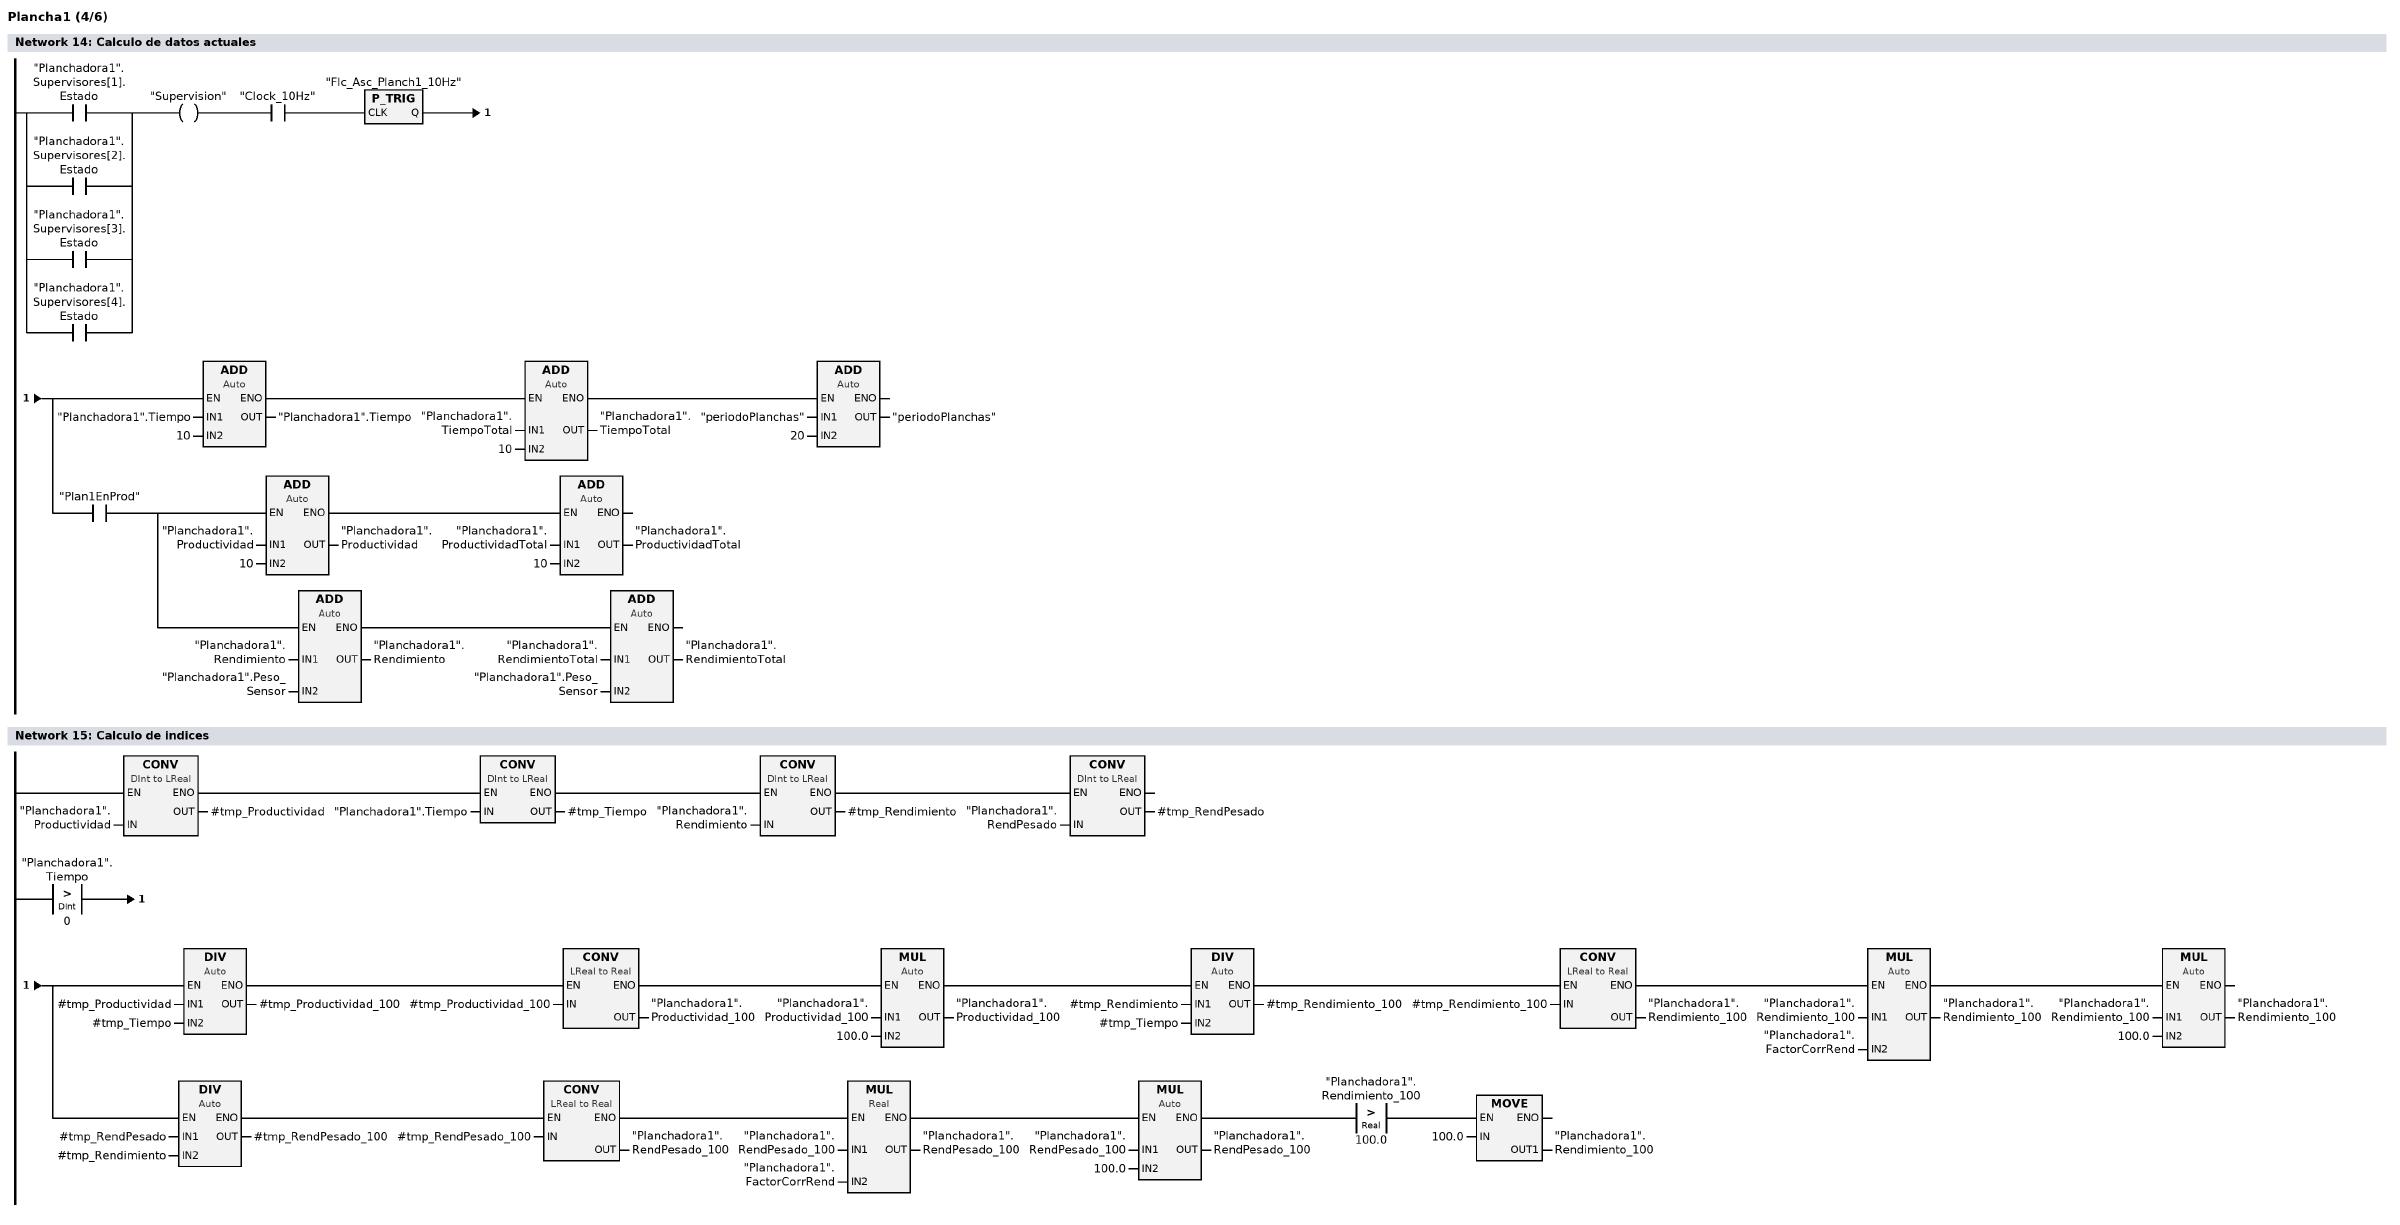
   RUNG wire#powerrail
      Contact( "Planchadora1".Supervisores[1].Estado )
      wire#w1
      Coil( "Supervision" )
      Contact( "Clock_10Hz" )
      P_Trig( "Flc_Asc_Planch1_10Hz" )
      wire#w2
      { S7_GenerateENO := "TRUE" } Add(in1 := "Planchadora1".Tiempo, in2 := 10, out => "Planchadora1".Tiempo)
      { S7_GenerateENO := "TRUE" } Add(in1 := "Planchadora1".TiempoTotal, in2 := 10, out => "Planchadora1".TiempoTotal)
      { S7_GenerateENO := "TRUE" } Add(in1 := "periodoPlanchas", in2 := 20, out => "periodoPlanchas")
   END_RUNG
   RUNG wire#powerrail
      Contact( "Planchadora1".Supervisores[2].Estado )
   END_RUNG wire#w1
   RUNG wire#powerrail
      Contact( "Planchadora1".Supervisores[3].Estado )
   END_RUNG wire#w1
   RUNG wire#powerrail
      Contact( "Planchadora1".Supervisores[4].Estado )
   END_RUNG wire#w1
   RUNG wire#w2
      Contact( "Plan1EnProd" )
      wire#w3
      { S7_GenerateENO := "TRUE" } Add(in1 := "Planchadora1".Productividad, in2 := 10, out => "Planchadora1".Productividad)
      { S7_GenerateENO := "TRUE" } Add(in1 := "Planchadora1".ProductividadTotal, in2 := 10, out => "Planchadora1".ProductividadTotal)
   END_RUNG
   RUNG wire#w3
      { S7_GenerateENO := "TRUE" } Add(in1 := "Planchadora1".Rendimiento, in2 := "Planchadora1".Peso_Sensor, out => "Planchadora1".Rendimiento)
      { S7_GenerateENO := "TRUE" } Add(in1 := "Planchadora1".RendimientoTotal, in2 := "Planchadora1".Peso_Sensor, out => "Planchadora1".RendimientoTotal)
   END_RUNG
   // the same network as SCL:
   // ENO of a box is taken as its EN; it also drops when the box reports an error
   "Supervision" := "Planchadora1".Supervisores[1].Estado OR "Planchadora1".Supervisores[2].Estado OR "Planchadora1".Supervisores[3].Estado OR "Planchadora1".Supervisores[4].Estado;
   #_w1 := "Supervision" AND "Clock_10Hz";
   #_w2 := #_w1 AND NOT "Flc_Asc_Planch1_10Hz";   // rising edge
   "Flc_Asc_Planch1_10Hz" := #_w1;
   IF #_w2 THEN
       "Planchadora1".Tiempo := "Planchadora1".Tiempo + 10;
       "Planchadora1".TiempoTotal := "Planchadora1".TiempoTotal + 10;
       "periodoPlanchas" := "periodoPlanchas" + 20;
   END_IF;
   IF #_w2 AND "Plan1EnProd" THEN
       "Planchadora1".Productividad := "Planchadora1".Productividad + 10;
       "Planchadora1".ProductividadTotal := "Planchadora1".ProductividadTotal + 10;
       "Planchadora1".Rendimiento := "Planchadora1".Rendimiento + "Planchadora1".Peso_Sensor;
       "Planchadora1".RendimientoTotal := "Planchadora1".RendimientoTotal + "Planchadora1".Peso_Sensor;
   END_IF;
END_REGION

REGION Network 15: Calculo de indices
   RUNG wire#powerrail
      { S7_Templates := "[SrcType := DInt, DestType := LReal]"; S7_GenerateENO := "TRUE" } Convert(in := "Planchadora1".Productividad, out => #tmp_Productividad)
      { S7_Templates := "[SrcType := DInt, DestType := LReal]"; S7_GenerateENO := "TRUE" } Convert(in := "Planchadora1".Tiempo, out => #tmp_Tiempo)
      { S7_Templates := "[SrcType := DInt, DestType := LReal]"; S7_GenerateENO := "TRUE" } Convert(in := "Planchadora1".Rendimiento, out => #tmp_Rendimiento)
      { S7_Templates := "[SrcType := DInt, DestType := LReal]"; S7_GenerateENO := "TRUE" } Convert(in := "Planchadora1".RendPesado, out => #tmp_RendPesado)
   END_RUNG
   RUNG wire#powerrail
      { S7_Templates := "SrcType := DInt" } GT_Contact(in1 := "Planchadora1".Tiempo, in2 := 0)
      wire#w1
      { S7_GenerateENO := "TRUE" } Div(in1 := #tmp_Productividad, in2 := #tmp_Tiempo, out => #tmp_Productividad_100)
      { S7_Templates := "[SrcType := LReal, DestType := Real]"; S7_GenerateENO := "TRUE" } Convert(in := #tmp_Productividad_100, out => "Planchadora1".Productividad_100)
      { S7_GenerateENO := "TRUE" } Mul(in1 := "Planchadora1".Productividad_100, in2 := 100.0, out => "Planchadora1".Productividad_100)
      { S7_GenerateENO := "TRUE" } Div(in1 := #tmp_Rendimiento, in2 := #tmp_Tiempo, out => #tmp_Rendimiento_100)
      { S7_Templates := "[SrcType := LReal, DestType := Real]"; S7_GenerateENO := "TRUE" } Convert(in := #tmp_Rendimiento_100, out => "Planchadora1".Rendimiento_100)
      { S7_GenerateENO := "TRUE" } Mul(in1 := "Planchadora1".Rendimiento_100, in2 := "Planchadora1".FactorCorrRend, out => "Planchadora1".Rendimiento_100)
      { S7_GenerateENO := "TRUE" } Mul(in1 := "Planchadora1".Rendimiento_100, in2 := 100.0, out => "Planchadora1".Rendimiento_100)
   END_RUNG
   RUNG wire#w1
      { S7_GenerateENO := "TRUE" } Div(in1 := #tmp_RendPesado, in2 := #tmp_Rendimiento, out => #tmp_RendPesado_100)
      { S7_Templates := "[SrcType := LReal, DestType := Real]"; S7_GenerateENO := "TRUE" } Convert(in := #tmp_RendPesado_100, out => "Planchadora1".RendPesado_100)
      { S7_Templates := "SrcType := Real"; S7_GenerateENO := "TRUE" } Mul(in1 := "Planchadora1".RendPesado_100, in2 := "Planchadora1".FactorCorrRend, out => "Planchadora1".RendPesado_100)
      { S7_GenerateENO := "TRUE" } Mul(in1 := "Planchadora1".RendPesado_100, in2 := 100.0, out => "Planchadora1".RendPesado_100)
      { S7_Templates := "SrcType := Real" } GT_Contact(in1 := "Planchadora1".Rendimiento_100, in2 := 100.0)
      { S7_GenerateENO := "TRUE" } Move(in := 100.0, out1 => "Planchadora1".Rendimiento_100)
   END_RUNG
   // the same network as SCL:
   // ENO of a box is taken as its EN; it also drops when the box reports an error
   #tmp_Productividad := DINT_TO_LREAL("Planchadora1".Productividad);
   #tmp_Tiempo := DINT_TO_LREAL("Planchadora1".Tiempo);
   #tmp_Rendimiento := DINT_TO_LREAL("Planchadora1".Rendimiento);
   #tmp_RendPesado := DINT_TO_LREAL("Planchadora1".RendPesado);
   #_w1 := "Planchadora1".Tiempo > 0;
   IF #_w1 THEN
       #tmp_Productividad_100 := #tmp_Productividad / #tmp_Tiempo;
       "Planchadora1".Productividad_100 := LREAL_TO_REAL(#tmp_Productividad_100);
       "Planchadora1".Productividad_100 := "Planchadora1".Productividad_100 * 100.0;
       #tmp_Rendimiento_100 := #tmp_Rendimiento / #tmp_Tiempo;
       "Planchadora1".Rendimiento_100 := LREAL_TO_REAL(#tmp_Rendimiento_100);
       "Planchadora1".Rendimiento_100 := "Planchadora1".Rendimiento_100 * "Planchadora1".FactorCorrRend;
       "Planchadora1".Rendimiento_100 := "Planchadora1".Rendimiento_100 * 100.0;
       #tmp_RendPesado_100 := #tmp_RendPesado / #tmp_Rendimiento;
       "Planchadora1".RendPesado_100 := LREAL_TO_REAL(#tmp_RendPesado_100);
       "Planchadora1".RendPesado_100 := "Planchadora1".RendPesado_100 * "Planchadora1".FactorCorrRend;
       "Planchadora1".RendPesado_100 := "Planchadora1".RendPesado_100 * 100.0;
   END_IF;
   IF #_w1 AND ("Planchadora1".Rendimiento_100 > 100.0) THEN "Planchadora1".Rendimiento_100 := 100.0; END_IF;
END_REGION

REGION Network 16: Variable cada 15 Minutos
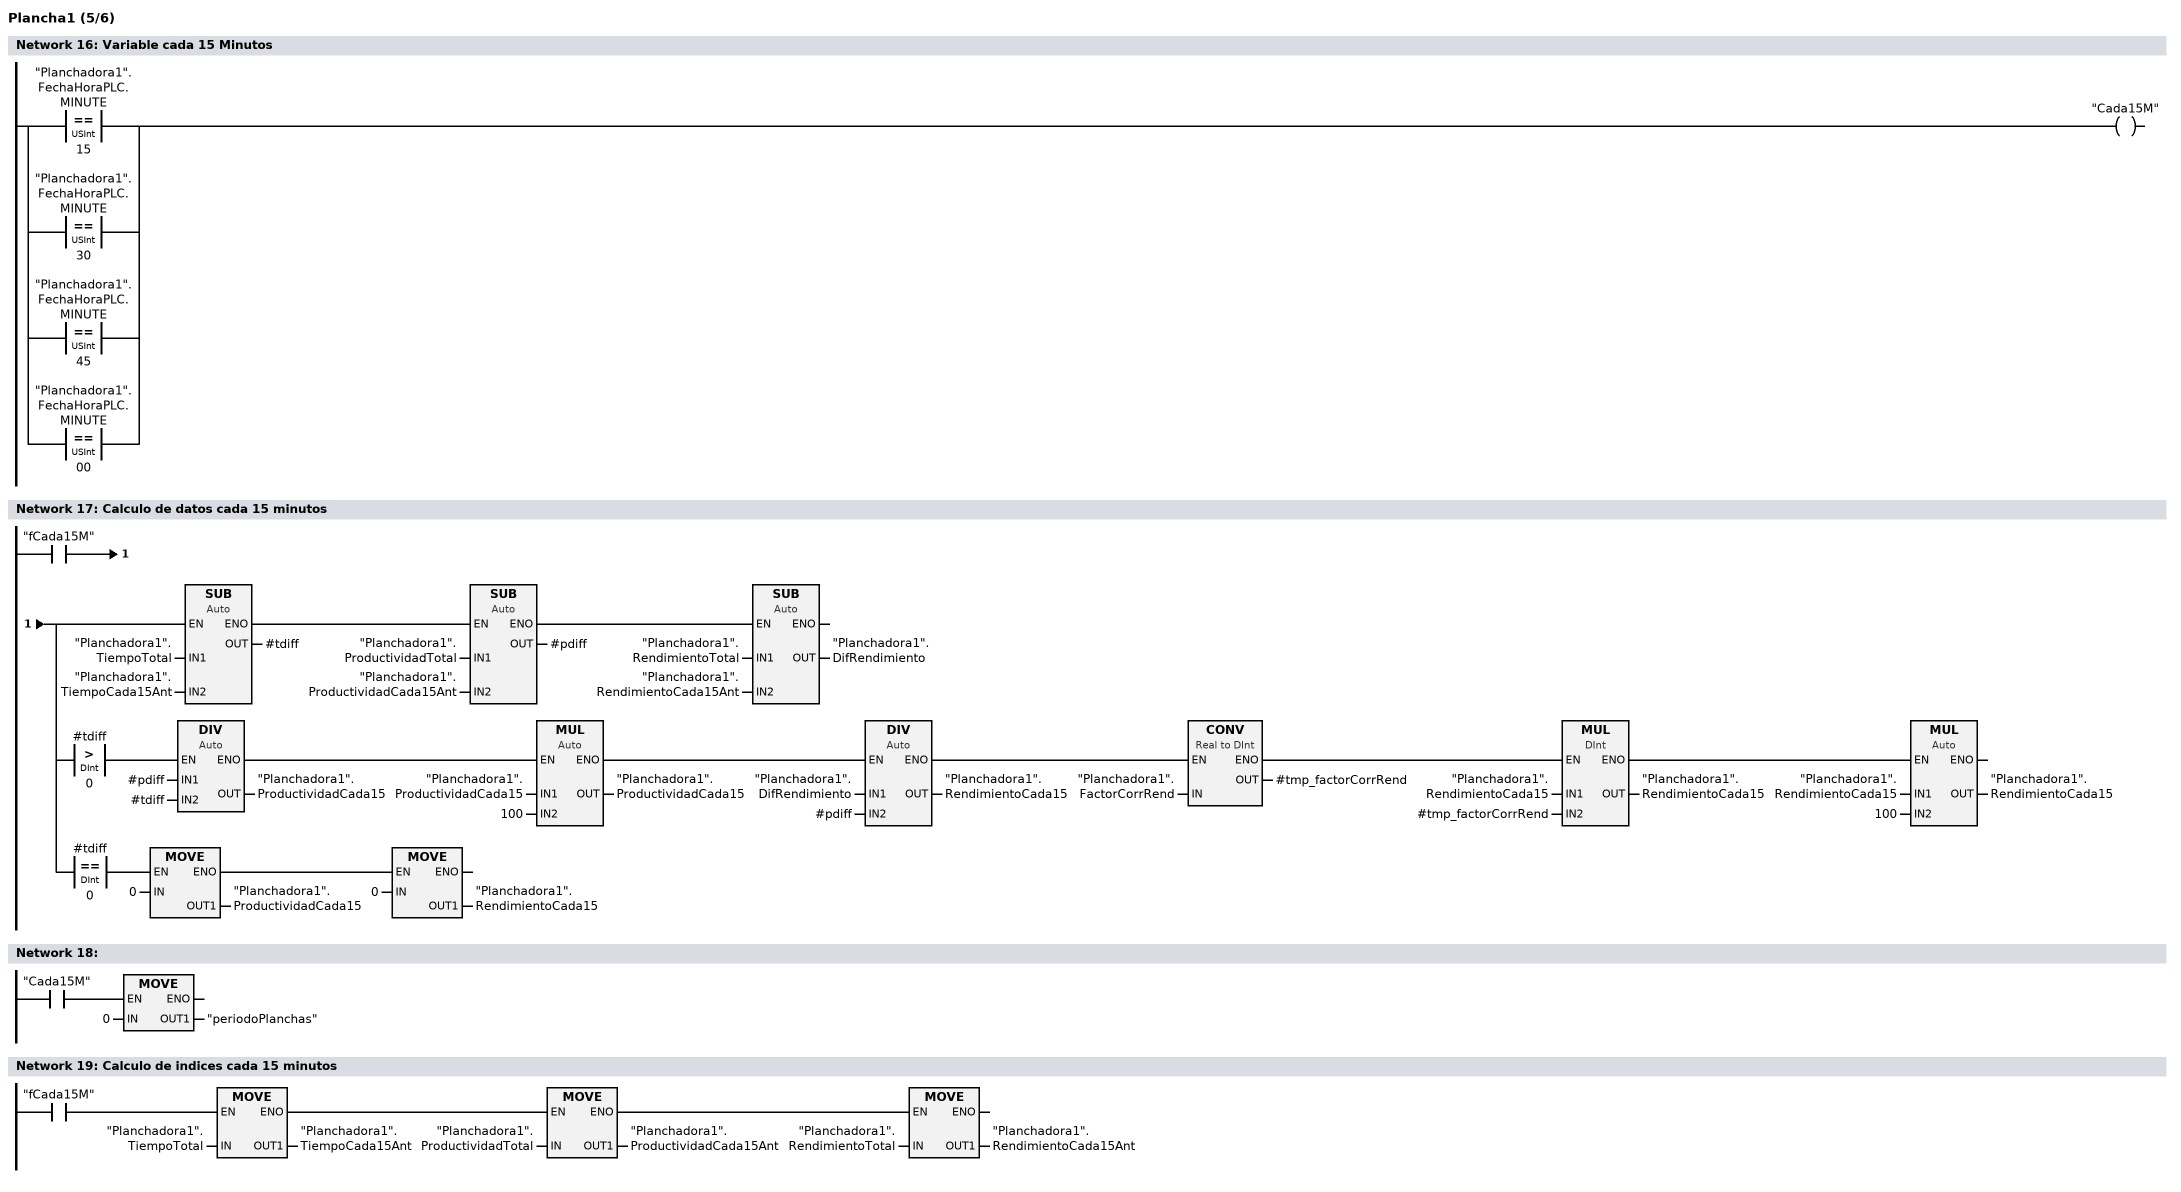
   RUNG wire#powerrail
      { S7_Templates := "SrcType := USInt" } EQ_Contact(in1 := "Planchadora1".FechaHoraPLC.MINUTE, in2 := 15)
      wire#w1
      Coil( "Cada15M" )
   END_RUNG
   RUNG wire#powerrail
      { S7_Templates := "SrcType := USInt" } EQ_Contact(in1 := "Planchadora1".FechaHoraPLC.MINUTE, in2 := 30)
   END_RUNG wire#w1
   RUNG wire#powerrail
      { S7_Templates := "SrcType := USInt" } EQ_Contact(in1 := "Planchadora1".FechaHoraPLC.MINUTE, in2 := 45)
   END_RUNG wire#w1
   RUNG wire#powerrail
      { S7_Templates := "SrcType := USInt" } EQ_Contact(in1 := "Planchadora1".FechaHoraPLC.MINUTE, in2 := 00)
   END_RUNG wire#w1
   // the same network as SCL:
   "Cada15M" := ("Planchadora1".FechaHoraPLC.MINUTE = 15) OR ("Planchadora1".FechaHoraPLC.MINUTE = 30) OR ("Planchadora1".FechaHoraPLC.MINUTE = 45) OR ("Planchadora1".FechaHoraPLC.MINUTE = 00);
END_REGION

REGION Network 17: Calculo de datos cada 15 minutos
   RUNG wire#powerrail
      Contact( "fCada15M" )
      wire#w1
      { S7_GenerateENO := "TRUE" } Sub(in1 := "Planchadora1".TiempoTotal, in2 := "Planchadora1".TiempoCada15Ant, out => #tdiff)
      { S7_GenerateENO := "TRUE" } Sub(in1 := "Planchadora1".ProductividadTotal, in2 := "Planchadora1".ProductividadCada15Ant, out => #pdiff)
      { S7_GenerateENO := "TRUE" } Sub(in1 := "Planchadora1".RendimientoTotal, in2 := "Planchadora1".RendimientoCada15Ant, out => "Planchadora1".DifRendimiento)
   END_RUNG
   RUNG wire#w1
      { S7_Templates := "SrcType := DInt" } GT_Contact(in1 := #tdiff, in2 := 0)
      { S7_GenerateENO := "TRUE" } Div(in1 := #pdiff, in2 := #tdiff, out => "Planchadora1".ProductividadCada15)
      { S7_GenerateENO := "TRUE" } Mul(in1 := "Planchadora1".ProductividadCada15, in2 := 100, out => "Planchadora1".ProductividadCada15)
      { S7_GenerateENO := "TRUE" } Div(in1 := "Planchadora1".DifRendimiento, in2 := #pdiff, out => "Planchadora1".RendimientoCada15)
      { S7_Templates := "[SrcType := Real, DestType := DInt]"; S7_GenerateENO := "TRUE" } Convert(in := "Planchadora1".FactorCorrRend, out => #tmp_factorCorrRend)
      { S7_Templates := "SrcType := DInt"; S7_GenerateENO := "TRUE" } Mul(in1 := "Planchadora1".RendimientoCada15, in2 := #tmp_factorCorrRend, out => "Planchadora1".RendimientoCada15)
      { S7_GenerateENO := "TRUE" } Mul(in1 := "Planchadora1".RendimientoCada15, in2 := 100, out => "Planchadora1".RendimientoCada15)
   END_RUNG
   RUNG wire#w1
      { S7_Templates := "SrcType := DInt" } EQ_Contact(in1 := #tdiff, in2 := 0)
      { S7_GenerateENO := "TRUE" } Move(in := 0, out1 => "Planchadora1".ProductividadCada15)
      { S7_GenerateENO := "TRUE" } Move(in := 0, out1 => "Planchadora1".RendimientoCada15)
   END_RUNG
   // the same network as SCL:
   // ENO of a box is taken as its EN; it also drops when the box reports an error
   IF "fCada15M" THEN
       #tdiff := "Planchadora1".TiempoTotal - "Planchadora1".TiempoCada15Ant;
       #pdiff := "Planchadora1".ProductividadTotal - "Planchadora1".ProductividadCada15Ant;
       "Planchadora1".DifRendimiento := "Planchadora1".RendimientoTotal - "Planchadora1".RendimientoCada15Ant;
   END_IF;
   IF "fCada15M" AND (#tdiff > 0) THEN
       "Planchadora1".ProductividadCada15 := #pdiff / #tdiff;
       "Planchadora1".ProductividadCada15 := "Planchadora1".ProductividadCada15 * 100;
       "Planchadora1".RendimientoCada15 := "Planchadora1".DifRendimiento / #pdiff;
       #tmp_factorCorrRend := REAL_TO_DINT("Planchadora1".FactorCorrRend);
       "Planchadora1".RendimientoCada15 := "Planchadora1".RendimientoCada15 * #tmp_factorCorrRend;
       "Planchadora1".RendimientoCada15 := "Planchadora1".RendimientoCada15 * 100;
   END_IF;
   IF "fCada15M" AND (#tdiff = 0) THEN
       "Planchadora1".ProductividadCada15 := 0;
       "Planchadora1".RendimientoCada15 := 0;
   END_IF;
END_REGION

REGION Network 18
   RUNG wire#powerrail
      Contact( "Cada15M" )
      { S7_GenerateENO := "TRUE" } Move(in := 0, out1 => "periodoPlanchas")
   END_RUNG
   // the same network as SCL:
   IF "Cada15M" THEN "periodoPlanchas" := 0; END_IF;
END_REGION

REGION Network 19: Calculo de indices cada 15 minutos
   RUNG wire#powerrail
      Contact( "fCada15M" )
      { S7_GenerateENO := "TRUE" } Move(in := "Planchadora1".TiempoTotal, out1 => "Planchadora1".TiempoCada15Ant)
      { S7_GenerateENO := "TRUE" } Move(in := "Planchadora1".ProductividadTotal, out1 => "Planchadora1".ProductividadCada15Ant)
      { S7_GenerateENO := "TRUE" } Move(in := "Planchadora1".RendimientoTotal, out1 => "Planchadora1".RendimientoCada15Ant)
   END_RUNG
   // the same network as SCL:
   // ENO of a box is taken as its EN; it also drops when the box reports an error
   IF "fCada15M" THEN
       "Planchadora1".TiempoCada15Ant := "Planchadora1".TiempoTotal;
       "Planchadora1".ProductividadCada15Ant := "Planchadora1".ProductividadTotal;
       "Planchadora1".RendimientoCada15Ant := "Planchadora1".RendimientoTotal;
   END_IF;
END_REGION

REGION Network 20: Definición de factor de Rendimiento
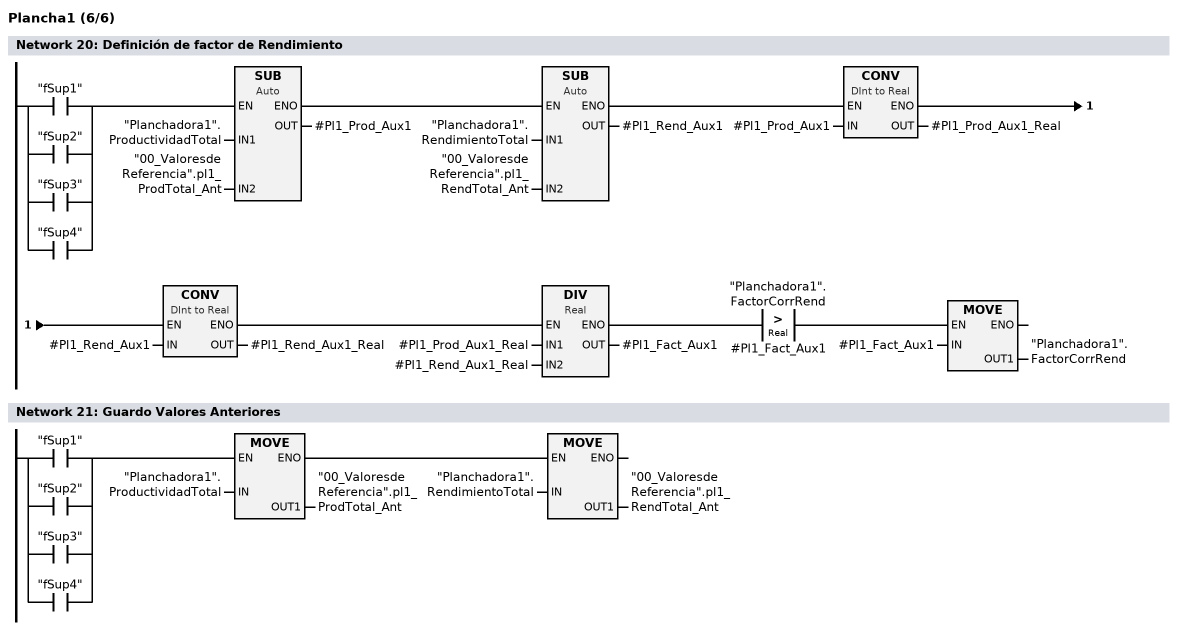
   RUNG wire#powerrail
      Contact( "fSup1" )
      wire#w1
      { S7_GenerateENO := "TRUE" } Sub(in1 := "Planchadora1".ProductividadTotal, in2 := "00_ValoresdeReferencia".pl1_ProdTotal_Ant, out => #Pl1_Prod_Aux1)
      { S7_GenerateENO := "TRUE" } Sub(in1 := "Planchadora1".RendimientoTotal, in2 := "00_ValoresdeReferencia".pl1_RendTotal_Ant, out => #Pl1_Rend_Aux1)
      { S7_Templates := "[SrcType := DInt, DestType := Real]"; S7_GenerateENO := "TRUE" } Convert(in := #Pl1_Prod_Aux1, out => #Pl1_Prod_Aux1_Real)
      { S7_Templates := "[SrcType := DInt, DestType := Real]"; S7_GenerateENO := "TRUE" } Convert(in := #Pl1_Rend_Aux1, out => #Pl1_Rend_Aux1_Real)
      { S7_Templates := "SrcType := Real"; S7_GenerateENO := "TRUE" } Div(in1 := #Pl1_Prod_Aux1_Real, in2 := #Pl1_Rend_Aux1_Real, out => #Pl1_Fact_Aux1)
      { S7_Templates := "SrcType := Real" } GT_Contact(in1 := "Planchadora1".FactorCorrRend, in2 := #Pl1_Fact_Aux1)
      { S7_GenerateENO := "TRUE" } Move(in := #Pl1_Fact_Aux1, out1 => "Planchadora1".FactorCorrRend)
   END_RUNG
   RUNG wire#powerrail
      Contact( "fSup2" )
   END_RUNG wire#w1
   RUNG wire#powerrail
      Contact( "fSup3" )
   END_RUNG wire#w1
   RUNG wire#powerrail
      Contact( "fSup4" )
   END_RUNG wire#w1
   // the same network as SCL:
   // ENO of a box is taken as its EN; it also drops when the box reports an error
   #_w1 := "fSup1" OR "fSup2" OR "fSup3" OR "fSup4";
   IF #_w1 THEN
       #Pl1_Prod_Aux1 := "Planchadora1".ProductividadTotal - "00_ValoresdeReferencia".pl1_ProdTotal_Ant;
       #Pl1_Rend_Aux1 := "Planchadora1".RendimientoTotal - "00_ValoresdeReferencia".pl1_RendTotal_Ant;
       #Pl1_Prod_Aux1_Real := DINT_TO_REAL(#Pl1_Prod_Aux1);
       #Pl1_Rend_Aux1_Real := DINT_TO_REAL(#Pl1_Rend_Aux1);
       #Pl1_Fact_Aux1 := #Pl1_Prod_Aux1_Real / #Pl1_Rend_Aux1_Real;
   END_IF;
   IF #_w1 AND ("Planchadora1".FactorCorrRend > #Pl1_Fact_Aux1) THEN
       "Planchadora1".FactorCorrRend := #Pl1_Fact_Aux1;
   END_IF;
END_REGION

REGION Network 21: Guardo Valores Anteriores
   RUNG wire#powerrail
      Contact( "fSup1" )
      wire#w1
      { S7_GenerateENO := "TRUE" } Move(in := "Planchadora1".ProductividadTotal, out1 => "00_ValoresdeReferencia".pl1_ProdTotal_Ant)
      { S7_GenerateENO := "TRUE" } Move(in := "Planchadora1".RendimientoTotal, out1 => "00_ValoresdeReferencia".pl1_RendTotal_Ant)
   END_RUNG
   RUNG wire#powerrail
      Contact( "fSup2" )
   END_RUNG wire#w1
   RUNG wire#powerrail
      Contact( "fSup3" )
   END_RUNG wire#w1
   RUNG wire#powerrail
      Contact( "fSup4" )
   END_RUNG wire#w1
   // the same network as SCL:
   // ENO of a box is taken as its EN; it also drops when the box reports an error
   IF "fSup1" OR "fSup2" OR "fSup3" OR "fSup4" THEN
       "00_ValoresdeReferencia".pl1_ProdTotal_Ant := "Planchadora1".ProductividadTotal;
       "00_ValoresdeReferencia".pl1_RendTotal_Ant := "Planchadora1".RendimientoTotal;
   END_IF;
END_REGION
END_FUNCTION

FUNCTION "Plancha2" : Void   // FC3, LAD
{ S7_Optimized_Access := 'FALSE' }
VERSION : 0.1
   VAR_TEMP
      rdiff : DInt;
      pdiff : DInt;
      tdiff : DInt;
      Temp_2 : Bool;
      tmp_Productividad_100 : LReal;
      "tmp_.Rendimiento_100" : LReal;
      tmp_RendPesado_100 : LReal;
      tmp_ProductividadCada15 : LReal;
      tmp_Productividad : LReal;
      tmp_Tiempo : LReal;
      tmp_RendPesado : LReal;
      tmp_Rendimiento : LReal;
      Pl2_Prod_Aux1 : DInt;
      Pl2_Rend_Aux1 : DInt;
      Pl2_Fact_Aux1 : Real;
      Pl2_Prod_Aux1_Real : Real;
      Pl2_Rend_Aux1_Real : Real;
      tmp_factorCorrRend : DInt;
   END_VAR
   VAR_TEMP   // added for the SCL form of the ladder/FBD networks
      _w1 : Bool;
      _w2 : Bool;
   END_VAR
BEGIN

REGION Network 1: Inversión de Señal de Sensores
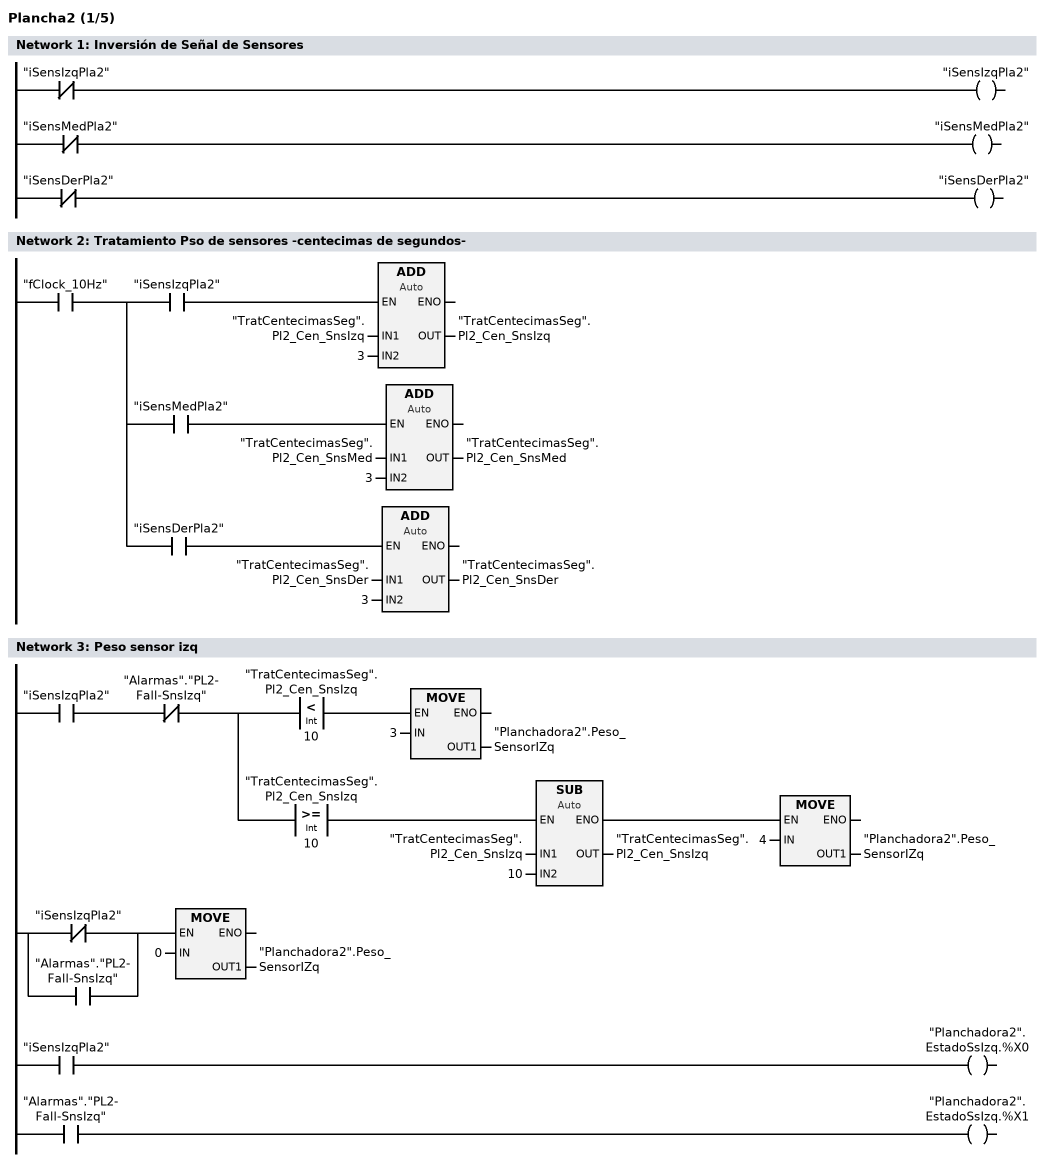
   RUNG wire#powerrail
      I_Contact( "iSensIzqPla2" )
      Coil( "iSensIzqPla2" )
   END_RUNG
   RUNG wire#powerrail
      I_Contact( "iSensMedPla2" )
      Coil( "iSensMedPla2" )
   END_RUNG
   RUNG wire#powerrail
      I_Contact( "iSensDerPla2" )
      Coil( "iSensDerPla2" )
   END_RUNG
   // the same network as SCL:
   "iSensIzqPla2" := NOT "iSensIzqPla2";
   "iSensMedPla2" := NOT "iSensMedPla2";
   "iSensDerPla2" := NOT "iSensDerPla2";
END_REGION

REGION Network 2: Tratamiento Pso de sensores -centecimas de segundos-
   RUNG wire#powerrail
      Contact( "fClock_10Hz" )
      wire#w1
      Contact( "iSensIzqPla2" )
      { S7_GenerateENO := "TRUE" } Add(in1 := "TratCentecimasSeg".Pl2_Cen_SnsIzq, in2 := 3, out => "TratCentecimasSeg".Pl2_Cen_SnsIzq)
   END_RUNG
   RUNG wire#w1
      Contact( "iSensMedPla2" )
      { S7_GenerateENO := "TRUE" } Add(in1 := "TratCentecimasSeg".Pl2_Cen_SnsMed, in2 := 3, out => "TratCentecimasSeg".Pl2_Cen_SnsMed)
   END_RUNG
   RUNG wire#w1
      Contact( "iSensDerPla2" )
      { S7_GenerateENO := "TRUE" } Add(in1 := "TratCentecimasSeg".Pl2_Cen_SnsDer, in2 := 3, out => "TratCentecimasSeg".Pl2_Cen_SnsDer)
   END_RUNG
   // the same network as SCL:
   IF "fClock_10Hz" AND "iSensIzqPla2" THEN
       "TratCentecimasSeg".Pl2_Cen_SnsIzq := "TratCentecimasSeg".Pl2_Cen_SnsIzq + 3;
   END_IF;
   IF "fClock_10Hz" AND "iSensMedPla2" THEN
       "TratCentecimasSeg".Pl2_Cen_SnsMed := "TratCentecimasSeg".Pl2_Cen_SnsMed + 3;
   END_IF;
   IF "fClock_10Hz" AND "iSensDerPla2" THEN
       "TratCentecimasSeg".Pl2_Cen_SnsDer := "TratCentecimasSeg".Pl2_Cen_SnsDer + 3;
   END_IF;
END_REGION

REGION Network 3: Peso sensor izq
   RUNG wire#powerrail
      Contact( "iSensIzqPla2" )
      I_Contact( "Alarmas"."PL2-Fall-SnsIzq" )
      wire#w1
      { S7_Templates := "SrcType := Int" } LT_Contact(in1 := "TratCentecimasSeg".Pl2_Cen_SnsIzq, in2 := 10)
      { S7_GenerateENO := "TRUE" } Move(in := 3, out1 => "Planchadora2".Peso_SensorIZq)
   END_RUNG
   RUNG wire#w1
      { S7_Templates := "SrcType := Int" } GE_Contact(in1 := "TratCentecimasSeg".Pl2_Cen_SnsIzq, in2 := 10)
      { S7_GenerateENO := "TRUE" } Sub(in1 := "TratCentecimasSeg".Pl2_Cen_SnsIzq, in2 := 10, out => "TratCentecimasSeg".Pl2_Cen_SnsIzq)
      { S7_GenerateENO := "TRUE" } Move(in := 4, out1 => "Planchadora2".Peso_SensorIZq)
   END_RUNG
   RUNG wire#powerrail
      I_Contact( "iSensIzqPla2" )
      wire#w2
      { S7_GenerateENO := "TRUE" } Move(in := 0, out1 => "Planchadora2".Peso_SensorIZq)
   END_RUNG
   RUNG wire#powerrail
      Contact( "Alarmas"."PL2-Fall-SnsIzq" )
   END_RUNG wire#w2
   RUNG wire#powerrail
      Contact( "iSensIzqPla2" )
      Coil( "Planchadora2".EstadoSsIzq.%X0 )
   END_RUNG
   RUNG wire#powerrail
      Contact( "Alarmas"."PL2-Fall-SnsIzq" )
      Coil( "Planchadora2".EstadoSsIzq.%X1 )
   END_RUNG
   // the same network as SCL:
   // ENO of a box is taken as its EN; it also drops when the box reports an error
   #_w1 := "iSensIzqPla2" AND NOT "Alarmas"."PL2-Fall-SnsIzq";
   IF #_w1 AND ("TratCentecimasSeg".Pl2_Cen_SnsIzq < 10) THEN "Planchadora2".Peso_SensorIZq := 3; END_IF;
   #_w2 := #_w1 AND ("TratCentecimasSeg".Pl2_Cen_SnsIzq >= 10);
   IF #_w2 THEN
       "TratCentecimasSeg".Pl2_Cen_SnsIzq := "TratCentecimasSeg".Pl2_Cen_SnsIzq - 10;
       "Planchadora2".Peso_SensorIZq := 4;
   END_IF;
   IF NOT "iSensIzqPla2" OR "Alarmas"."PL2-Fall-SnsIzq" THEN "Planchadora2".Peso_SensorIZq := 0; END_IF;
   "Planchadora2".EstadoSsIzq.%X0 := "iSensIzqPla2";
   "Planchadora2".EstadoSsIzq.%X1 := "Alarmas"."PL2-Fall-SnsIzq";
END_REGION

REGION Network 4: Peso sensor derecho
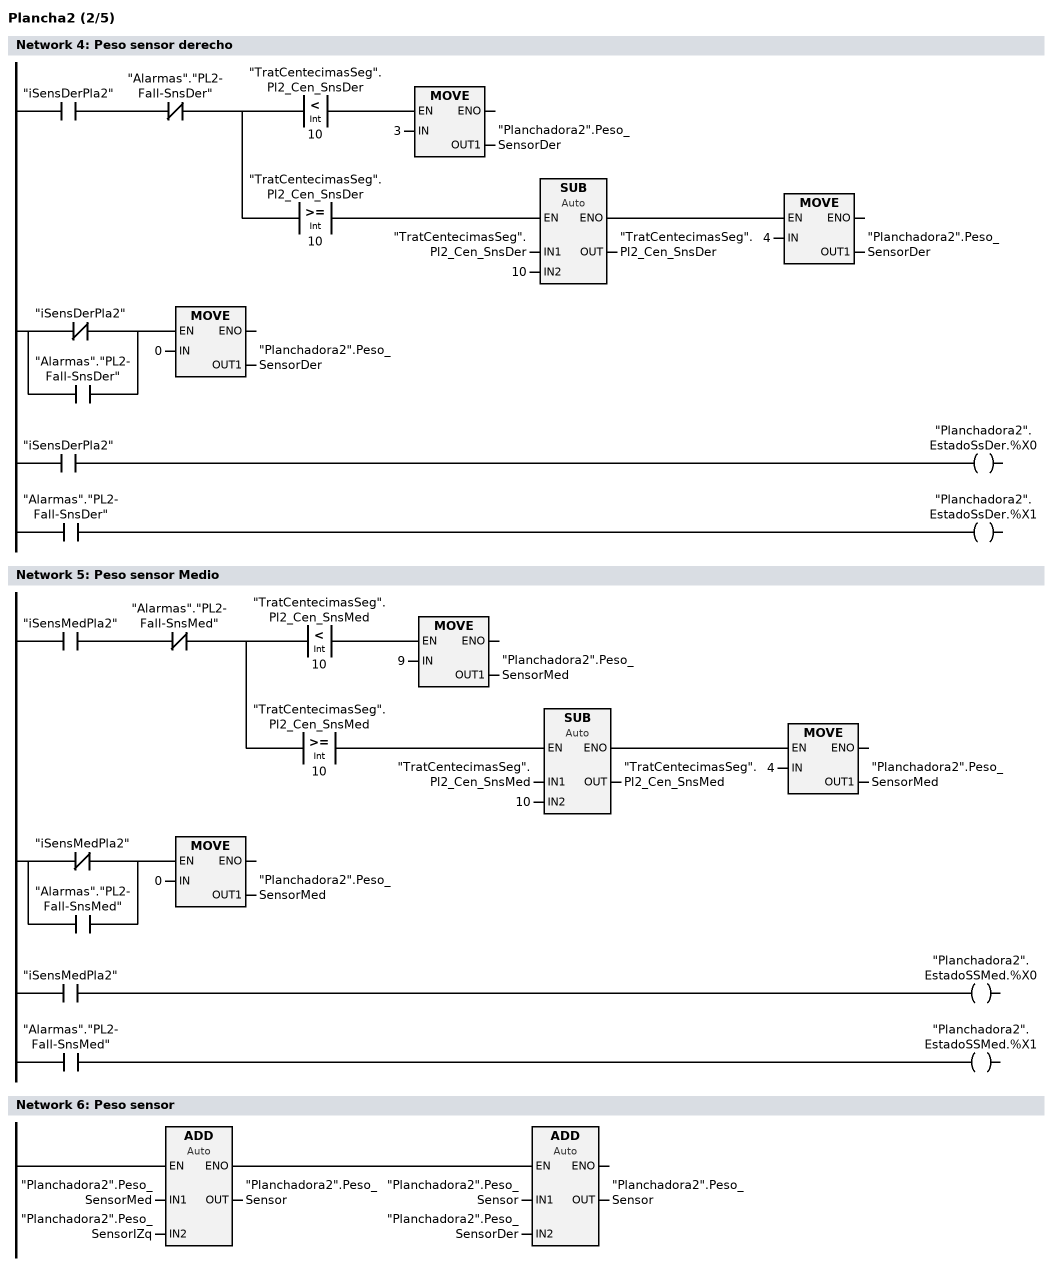
   RUNG wire#powerrail
      Contact( "iSensDerPla2" )
      I_Contact( "Alarmas"."PL2-Fall-SnsDer" )
      wire#w1
      { S7_Templates := "SrcType := Int" } LT_Contact(in1 := "TratCentecimasSeg".Pl2_Cen_SnsDer, in2 := 10)
      { S7_GenerateENO := "TRUE" } Move(in := 3, out1 => "Planchadora2".Peso_SensorDer)
   END_RUNG
   RUNG wire#w1
      { S7_Templates := "SrcType := Int" } GE_Contact(in1 := "TratCentecimasSeg".Pl2_Cen_SnsDer, in2 := 10)
      { S7_GenerateENO := "TRUE" } Sub(in1 := "TratCentecimasSeg".Pl2_Cen_SnsDer, in2 := 10, out => "TratCentecimasSeg".Pl2_Cen_SnsDer)
      { S7_GenerateENO := "TRUE" } Move(in := 4, out1 => "Planchadora2".Peso_SensorDer)
   END_RUNG
   RUNG wire#powerrail
      I_Contact( "iSensDerPla2" )
      wire#w2
      { S7_GenerateENO := "TRUE" } Move(in := 0, out1 => "Planchadora2".Peso_SensorDer)
   END_RUNG
   RUNG wire#powerrail
      Contact( "Alarmas"."PL2-Fall-SnsDer" )
   END_RUNG wire#w2
   RUNG wire#powerrail
      Contact( "iSensDerPla2" )
      Coil( "Planchadora2".EstadoSsDer.%X0 )
   END_RUNG
   RUNG wire#powerrail
      Contact( "Alarmas"."PL2-Fall-SnsDer" )
      Coil( "Planchadora2".EstadoSsDer.%X1 )
   END_RUNG
   // the same network as SCL:
   // ENO of a box is taken as its EN; it also drops when the box reports an error
   #_w1 := "iSensDerPla2" AND NOT "Alarmas"."PL2-Fall-SnsDer";
   IF #_w1 AND ("TratCentecimasSeg".Pl2_Cen_SnsDer < 10) THEN "Planchadora2".Peso_SensorDer := 3; END_IF;
   #_w2 := #_w1 AND ("TratCentecimasSeg".Pl2_Cen_SnsDer >= 10);
   IF #_w2 THEN
       "TratCentecimasSeg".Pl2_Cen_SnsDer := "TratCentecimasSeg".Pl2_Cen_SnsDer - 10;
       "Planchadora2".Peso_SensorDer := 4;
   END_IF;
   IF NOT "iSensDerPla2" OR "Alarmas"."PL2-Fall-SnsDer" THEN "Planchadora2".Peso_SensorDer := 0; END_IF;
   "Planchadora2".EstadoSsDer.%X0 := "iSensDerPla2";
   "Planchadora2".EstadoSsDer.%X1 := "Alarmas"."PL2-Fall-SnsDer";
END_REGION

REGION Network 5: Peso sensor Medio
   RUNG wire#powerrail
      Contact( "iSensMedPla2" )
      I_Contact( "Alarmas"."PL2-Fall-SnsMed" )
      wire#w1
      { S7_Templates := "SrcType := Int" } LT_Contact(in1 := "TratCentecimasSeg".Pl2_Cen_SnsMed, in2 := 10)
      { S7_GenerateENO := "TRUE" } Move(in := 9, out1 => "Planchadora2".Peso_SensorMed)
   END_RUNG
   RUNG wire#w1
      { S7_Templates := "SrcType := Int" } GE_Contact(in1 := "TratCentecimasSeg".Pl2_Cen_SnsMed, in2 := 10)
      { S7_GenerateENO := "TRUE" } Sub(in1 := "TratCentecimasSeg".Pl2_Cen_SnsMed, in2 := 10, out => "TratCentecimasSeg".Pl2_Cen_SnsMed)
      { S7_GenerateENO := "TRUE" } Move(in := 4, out1 => "Planchadora2".Peso_SensorMed)
   END_RUNG
   RUNG wire#powerrail
      I_Contact( "iSensMedPla2" )
      wire#w2
      { S7_GenerateENO := "TRUE" } Move(in := 0, out1 => "Planchadora2".Peso_SensorMed)
   END_RUNG
   RUNG wire#powerrail
      Contact( "Alarmas"."PL2-Fall-SnsMed" )
   END_RUNG wire#w2
   RUNG wire#powerrail
      Contact( "iSensMedPla2" )
      Coil( "Planchadora2".EstadoSSMed.%X0 )
   END_RUNG
   RUNG wire#powerrail
      Contact( "Alarmas"."PL2-Fall-SnsMed" )
      Coil( "Planchadora2".EstadoSSMed.%X1 )
   END_RUNG
   // the same network as SCL:
   // ENO of a box is taken as its EN; it also drops when the box reports an error
   #_w1 := "iSensMedPla2" AND NOT "Alarmas"."PL2-Fall-SnsMed";
   IF #_w1 AND ("TratCentecimasSeg".Pl2_Cen_SnsMed < 10) THEN "Planchadora2".Peso_SensorMed := 9; END_IF;
   #_w2 := #_w1 AND ("TratCentecimasSeg".Pl2_Cen_SnsMed >= 10);
   IF #_w2 THEN
       "TratCentecimasSeg".Pl2_Cen_SnsMed := "TratCentecimasSeg".Pl2_Cen_SnsMed - 10;
       "Planchadora2".Peso_SensorMed := 4;
   END_IF;
   IF NOT "iSensMedPla2" OR "Alarmas"."PL2-Fall-SnsMed" THEN "Planchadora2".Peso_SensorMed := 0; END_IF;
   "Planchadora2".EstadoSSMed.%X0 := "iSensMedPla2";
   "Planchadora2".EstadoSSMed.%X1 := "Alarmas"."PL2-Fall-SnsMed";
END_REGION

REGION Network 6: Peso sensor
   RUNG wire#powerrail
      { S7_GenerateENO := "TRUE" } Add(in1 := "Planchadora2".Peso_SensorMed, in2 := "Planchadora2".Peso_SensorIZq, out => "Planchadora2".Peso_Sensor)
      { S7_GenerateENO := "TRUE" } Add(in1 := "Planchadora2".Peso_Sensor, in2 := "Planchadora2".Peso_SensorDer, out => "Planchadora2".Peso_Sensor)
   END_RUNG
   // the same network as SCL:
   // ENO of a box is taken as its EN; it also drops when the box reports an error
   "Planchadora2".Peso_Sensor := "Planchadora2".Peso_SensorMed + "Planchadora2".Peso_SensorIZq;
   "Planchadora2".Peso_Sensor := "Planchadora2".Peso_Sensor + "Planchadora2".Peso_SensorDer;
END_REGION

REGION Network 7: Plancha 2 produccion
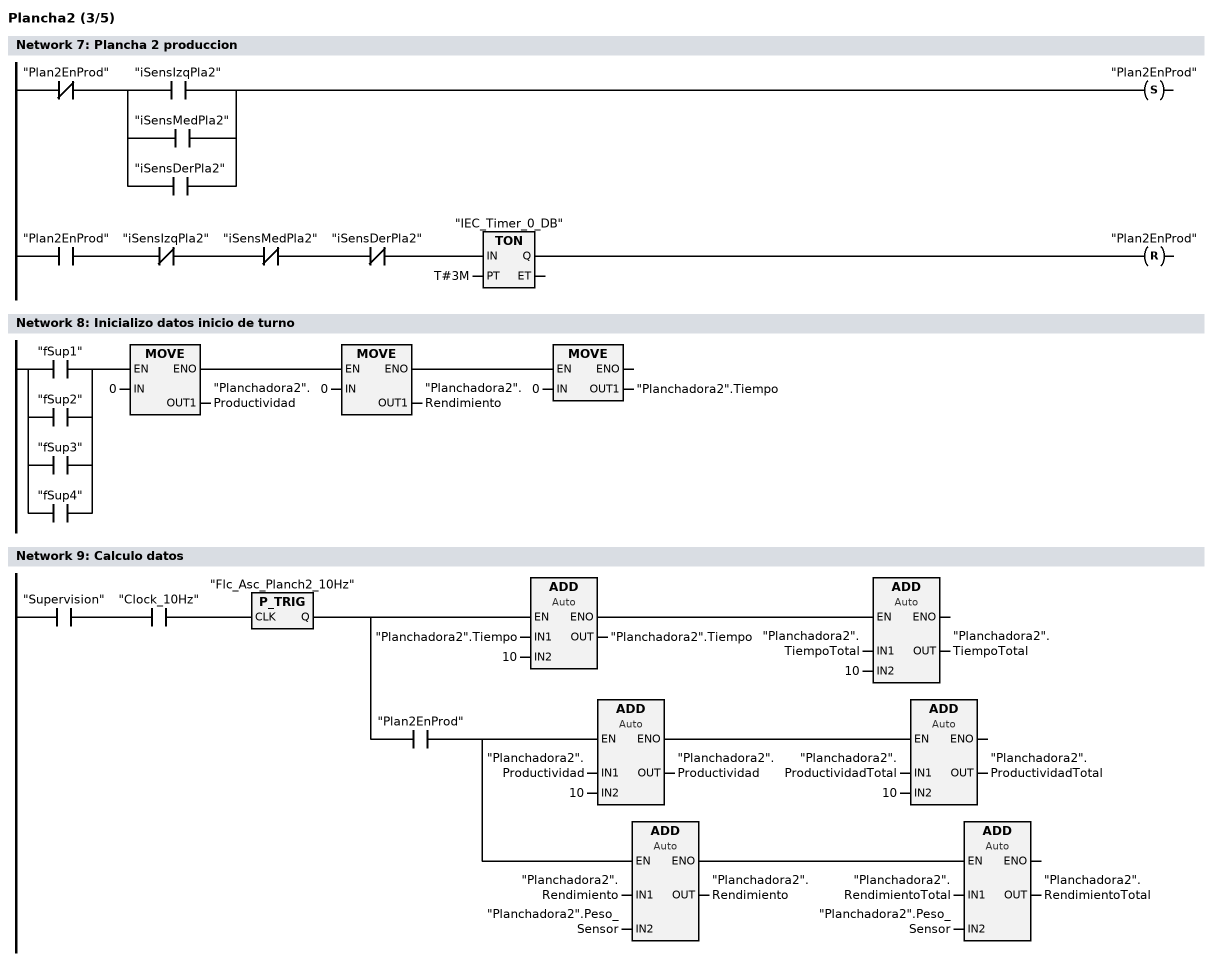
   IF NOT "Plan2EnProd" AND ("iSensIzqPla2" OR "iSensMedPla2" OR "iSensDerPla2") THEN
       "Plan2EnProd" := TRUE;
   END_IF;
   "IEC_Timer_0_DB".TON(IN := "Plan2EnProd" AND NOT "iSensIzqPla2" AND NOT "iSensMedPla2" AND NOT "iSensDerPla2",
                        PT := T#3M);
   IF "IEC_Timer_0_DB".Q THEN "Plan2EnProd" := FALSE; END_IF;
END_REGION

REGION Network 8: Inicializo datos inicio de turno
   RUNG wire#powerrail
      Contact( "fSup1" )
      wire#w1
      { S7_GenerateENO := "TRUE" } Move(in := 0, out1 => "Planchadora2".Productividad)
      { S7_GenerateENO := "TRUE" } Move(in := 0, out1 => "Planchadora2".Rendimiento)
      { S7_GenerateENO := "TRUE" } Move(in := 0, out1 => "Planchadora2".Tiempo)
   END_RUNG
   RUNG wire#powerrail
      Contact( "fSup2" )
   END_RUNG wire#w1
   RUNG wire#powerrail
      Contact( "fSup3" )
   END_RUNG wire#w1
   RUNG wire#powerrail
      Contact( "fSup4" )
   END_RUNG wire#w1
   // the same network as SCL:
   // ENO of a box is taken as its EN; it also drops when the box reports an error
   IF "fSup1" OR "fSup2" OR "fSup3" OR "fSup4" THEN
       "Planchadora2".Productividad := 0;
       "Planchadora2".Rendimiento := 0;
       "Planchadora2".Tiempo := 0;
   END_IF;
END_REGION

REGION Network 9: Calculo datos
   RUNG wire#powerrail
      Contact( "Supervision" )
      Contact( "Clock_10Hz" )
      P_Trig( "Flc_Asc_Planch2_10Hz" )
      wire#w1
      { S7_GenerateENO := "TRUE" } Add(in1 := "Planchadora2".Tiempo, in2 := 10, out => "Planchadora2".Tiempo)
      { S7_GenerateENO := "TRUE" } Add(in1 := "Planchadora2".TiempoTotal, in2 := 10, out => "Planchadora2".TiempoTotal)
   END_RUNG
   RUNG wire#w1
      Contact( "Plan2EnProd" )
      wire#w2
      { S7_GenerateENO := "TRUE" } Add(in1 := "Planchadora2".Productividad, in2 := 10, out => "Planchadora2".Productividad)
      { S7_GenerateENO := "TRUE" } Add(in1 := "Planchadora2".ProductividadTotal, in2 := 10, out => "Planchadora2".ProductividadTotal)
   END_RUNG
   RUNG wire#w2
      { S7_GenerateENO := "TRUE" } Add(in1 := "Planchadora2".Rendimiento, in2 := "Planchadora2".Peso_Sensor, out => "Planchadora2".Rendimiento)
      { S7_GenerateENO := "TRUE" } Add(in1 := "Planchadora2".RendimientoTotal, in2 := "Planchadora2".Peso_Sensor, out => "Planchadora2".RendimientoTotal)
   END_RUNG
   // the same network as SCL:
   // ENO of a box is taken as its EN; it also drops when the box reports an error
   #_w1 := "Supervision" AND "Clock_10Hz";
   #_w2 := #_w1 AND NOT "Flc_Asc_Planch2_10Hz";   // rising edge
   "Flc_Asc_Planch2_10Hz" := #_w1;
   IF #_w2 THEN
       "Planchadora2".Tiempo := "Planchadora2".Tiempo + 10;
       "Planchadora2".TiempoTotal := "Planchadora2".TiempoTotal + 10;
   END_IF;
   IF #_w2 AND "Plan2EnProd" THEN
       "Planchadora2".Productividad := "Planchadora2".Productividad + 10;
       "Planchadora2".ProductividadTotal := "Planchadora2".ProductividadTotal + 10;
       "Planchadora2".Rendimiento := "Planchadora2".Rendimiento + "Planchadora2".Peso_Sensor;
       "Planchadora2".RendimientoTotal := "Planchadora2".RendimientoTotal + "Planchadora2".Peso_Sensor;
   END_IF;
END_REGION

REGION Network 10: Calculo indices
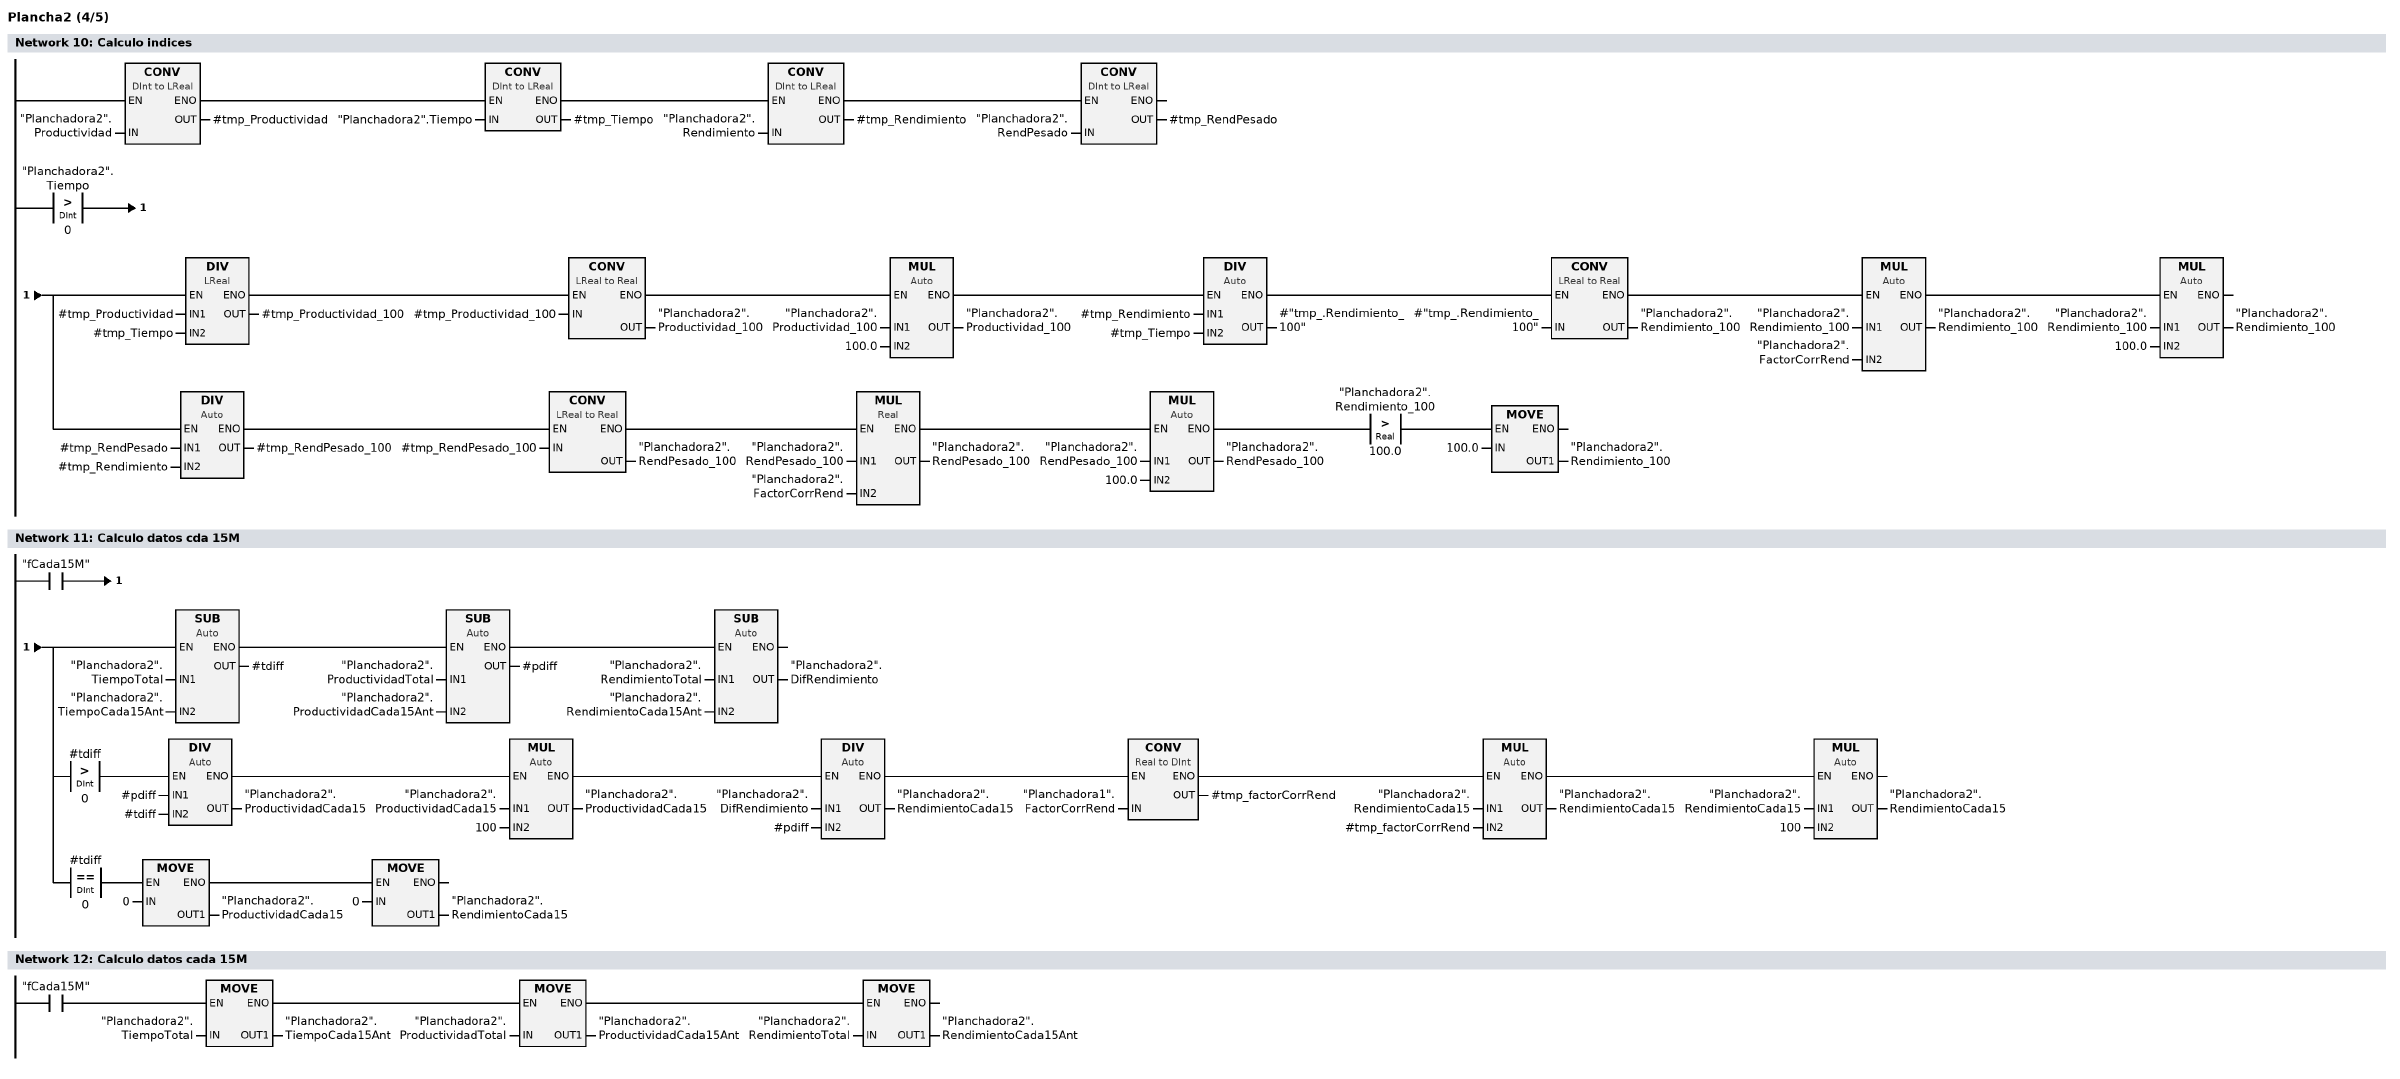
   RUNG wire#powerrail
      { S7_Templates := "[SrcType := DInt, DestType := LReal]"; S7_GenerateENO := "TRUE" } Convert(in := "Planchadora2".Productividad, out => #tmp_Productividad)
      { S7_Templates := "[SrcType := DInt, DestType := LReal]"; S7_GenerateENO := "TRUE" } Convert(in := "Planchadora2".Tiempo, out => #tmp_Tiempo)
      { S7_Templates := "[SrcType := DInt, DestType := LReal]"; S7_GenerateENO := "TRUE" } Convert(in := "Planchadora2".Rendimiento, out => #tmp_Rendimiento)
      { S7_Templates := "[SrcType := DInt, DestType := LReal]"; S7_GenerateENO := "TRUE" } Convert(in := "Planchadora2".RendPesado, out => #tmp_RendPesado)
   END_RUNG
   RUNG wire#powerrail
      { S7_Templates := "SrcType := DInt" } GT_Contact(in1 := "Planchadora2".Tiempo, in2 := 0)
      wire#w1
      { S7_Templates := "SrcType := LReal"; S7_GenerateENO := "TRUE" } Div(in1 := #tmp_Productividad, in2 := #tmp_Tiempo, out => #tmp_Productividad_100)
      { S7_Templates := "[SrcType := LReal, DestType := Real]"; S7_GenerateENO := "TRUE" } Convert(in := #tmp_Productividad_100, out => "Planchadora2".Productividad_100)
      { S7_GenerateENO := "TRUE" } Mul(in1 := "Planchadora2".Productividad_100, in2 := 100.0, out => "Planchadora2".Productividad_100)
      { S7_GenerateENO := "TRUE" } Div(in1 := #tmp_Rendimiento, in2 := #tmp_Tiempo, out => #"tmp_.Rendimiento_100")
      { S7_Templates := "[SrcType := LReal, DestType := Real]"; S7_GenerateENO := "TRUE" } Convert(in := #"tmp_.Rendimiento_100", out => "Planchadora2".Rendimiento_100)
      { S7_GenerateENO := "TRUE" } Mul(in1 := "Planchadora2".Rendimiento_100, in2 := "Planchadora2".FactorCorrRend, out => "Planchadora2".Rendimiento_100)
      { S7_GenerateENO := "TRUE" } Mul(in1 := "Planchadora2".Rendimiento_100, in2 := 100.0, out => "Planchadora2".Rendimiento_100)
   END_RUNG
   RUNG wire#w1
      { S7_GenerateENO := "TRUE" } Div(in1 := #tmp_RendPesado, in2 := #tmp_Rendimiento, out => #tmp_RendPesado_100)
      { S7_Templates := "[SrcType := LReal, DestType := Real]"; S7_GenerateENO := "TRUE" } Convert(in := #tmp_RendPesado_100, out => "Planchadora2".RendPesado_100)
      { S7_Templates := "SrcType := Real"; S7_GenerateENO := "TRUE" } Mul(in1 := "Planchadora2".RendPesado_100, in2 := "Planchadora2".FactorCorrRend, out => "Planchadora2".RendPesado_100)
      { S7_GenerateENO := "TRUE" } Mul(in1 := "Planchadora2".RendPesado_100, in2 := 100.0, out => "Planchadora2".RendPesado_100)
      { S7_Templates := "SrcType := Real" } GT_Contact(in1 := "Planchadora2".Rendimiento_100, in2 := 100.0)
      { S7_GenerateENO := "TRUE" } Move(in := 100.0, out1 => "Planchadora2".Rendimiento_100)
   END_RUNG
   // the same network as SCL:
   // ENO of a box is taken as its EN; it also drops when the box reports an error
   #tmp_Productividad := DINT_TO_LREAL("Planchadora2".Productividad);
   #tmp_Tiempo := DINT_TO_LREAL("Planchadora2".Tiempo);
   #tmp_Rendimiento := DINT_TO_LREAL("Planchadora2".Rendimiento);
   #tmp_RendPesado := DINT_TO_LREAL("Planchadora2".RendPesado);
   #_w1 := "Planchadora2".Tiempo > 0;
   IF #_w1 THEN
       #tmp_Productividad_100 := #tmp_Productividad / #tmp_Tiempo;
       "Planchadora2".Productividad_100 := LREAL_TO_REAL(#tmp_Productividad_100);
       "Planchadora2".Productividad_100 := "Planchadora2".Productividad_100 * 100.0;
       #"tmp_.Rendimiento_100" := #tmp_Rendimiento / #tmp_Tiempo;
       "Planchadora2".Rendimiento_100 := LREAL_TO_REAL(#"tmp_.Rendimiento_100");
       "Planchadora2".Rendimiento_100 := "Planchadora2".Rendimiento_100 * "Planchadora2".FactorCorrRend;
       "Planchadora2".Rendimiento_100 := "Planchadora2".Rendimiento_100 * 100.0;
       #tmp_RendPesado_100 := #tmp_RendPesado / #tmp_Rendimiento;
       "Planchadora2".RendPesado_100 := LREAL_TO_REAL(#tmp_RendPesado_100);
       "Planchadora2".RendPesado_100 := "Planchadora2".RendPesado_100 * "Planchadora2".FactorCorrRend;
       "Planchadora2".RendPesado_100 := "Planchadora2".RendPesado_100 * 100.0;
   END_IF;
   IF #_w1 AND ("Planchadora2".Rendimiento_100 > 100.0) THEN "Planchadora2".Rendimiento_100 := 100.0; END_IF;
END_REGION

REGION Network 11: Calculo datos cda 15M
   RUNG wire#powerrail
      Contact( "fCada15M" )
      wire#w1
      { S7_GenerateENO := "TRUE" } Sub(in1 := "Planchadora2".TiempoTotal, in2 := "Planchadora2".TiempoCada15Ant, out => #tdiff)
      { S7_GenerateENO := "TRUE" } Sub(in1 := "Planchadora2".ProductividadTotal, in2 := "Planchadora2".ProductividadCada15Ant, out => #pdiff)
      { S7_GenerateENO := "TRUE" } Sub(in1 := "Planchadora2".RendimientoTotal, in2 := "Planchadora2".RendimientoCada15Ant, out => "Planchadora2".DifRendimiento)
   END_RUNG
   RUNG wire#w1
      { S7_Templates := "SrcType := DInt" } GT_Contact(in1 := #tdiff, in2 := 0)
      { S7_GenerateENO := "TRUE" } Div(in1 := #pdiff, in2 := #tdiff, out => "Planchadora2".ProductividadCada15)
      { S7_GenerateENO := "TRUE" } Mul(in1 := "Planchadora2".ProductividadCada15, in2 := 100, out => "Planchadora2".ProductividadCada15)
      { S7_GenerateENO := "TRUE" } Div(in1 := "Planchadora2".DifRendimiento, in2 := #pdiff, out => "Planchadora2".RendimientoCada15)
      { S7_Templates := "[SrcType := Real, DestType := DInt]"; S7_GenerateENO := "TRUE" } Convert(in := "Planchadora1".FactorCorrRend, out => #tmp_factorCorrRend)
      { S7_GenerateENO := "TRUE" } Mul(in1 := "Planchadora2".RendimientoCada15, in2 := #tmp_factorCorrRend, out => "Planchadora2".RendimientoCada15)
      { S7_GenerateENO := "TRUE" } Mul(in1 := "Planchadora2".RendimientoCada15, in2 := 100, out => "Planchadora2".RendimientoCada15)
   END_RUNG
   RUNG wire#w1
      { S7_Templates := "SrcType := DInt" } EQ_Contact(in1 := #tdiff, in2 := 0)
      { S7_GenerateENO := "TRUE" } Move(in := 0, out1 => "Planchadora2".ProductividadCada15)
      { S7_GenerateENO := "TRUE" } Move(in := 0, out1 => "Planchadora2".RendimientoCada15)
   END_RUNG
   // the same network as SCL:
   // ENO of a box is taken as its EN; it also drops when the box reports an error
   IF "fCada15M" THEN
       #tdiff := "Planchadora2".TiempoTotal - "Planchadora2".TiempoCada15Ant;
       #pdiff := "Planchadora2".ProductividadTotal - "Planchadora2".ProductividadCada15Ant;
       "Planchadora2".DifRendimiento := "Planchadora2".RendimientoTotal - "Planchadora2".RendimientoCada15Ant;
   END_IF;
   IF "fCada15M" AND (#tdiff > 0) THEN
       "Planchadora2".ProductividadCada15 := #pdiff / #tdiff;
       "Planchadora2".ProductividadCada15 := "Planchadora2".ProductividadCada15 * 100;
       "Planchadora2".RendimientoCada15 := "Planchadora2".DifRendimiento / #pdiff;
       #tmp_factorCorrRend := REAL_TO_DINT("Planchadora1".FactorCorrRend);
       "Planchadora2".RendimientoCada15 := "Planchadora2".RendimientoCada15 * #tmp_factorCorrRend;
       "Planchadora2".RendimientoCada15 := "Planchadora2".RendimientoCada15 * 100;
   END_IF;
   IF "fCada15M" AND (#tdiff = 0) THEN
       "Planchadora2".ProductividadCada15 := 0;
       "Planchadora2".RendimientoCada15 := 0;
   END_IF;
END_REGION

REGION Network 12: Calculo datos cada 15M
   RUNG wire#powerrail
      Contact( "fCada15M" )
      { S7_GenerateENO := "TRUE" } Move(in := "Planchadora2".TiempoTotal, out1 => "Planchadora2".TiempoCada15Ant)
      { S7_GenerateENO := "TRUE" } Move(in := "Planchadora2".ProductividadTotal, out1 => "Planchadora2".ProductividadCada15Ant)
      { S7_GenerateENO := "TRUE" } Move(in := "Planchadora2".RendimientoTotal, out1 => "Planchadora2".RendimientoCada15Ant)
   END_RUNG
   // the same network as SCL:
   // ENO of a box is taken as its EN; it also drops when the box reports an error
   IF "fCada15M" THEN
       "Planchadora2".TiempoCada15Ant := "Planchadora2".TiempoTotal;
       "Planchadora2".ProductividadCada15Ant := "Planchadora2".ProductividadTotal;
       "Planchadora2".RendimientoCada15Ant := "Planchadora2".RendimientoTotal;
   END_IF;
END_REGION

REGION Network 13: Definición de factor de Rendimiento
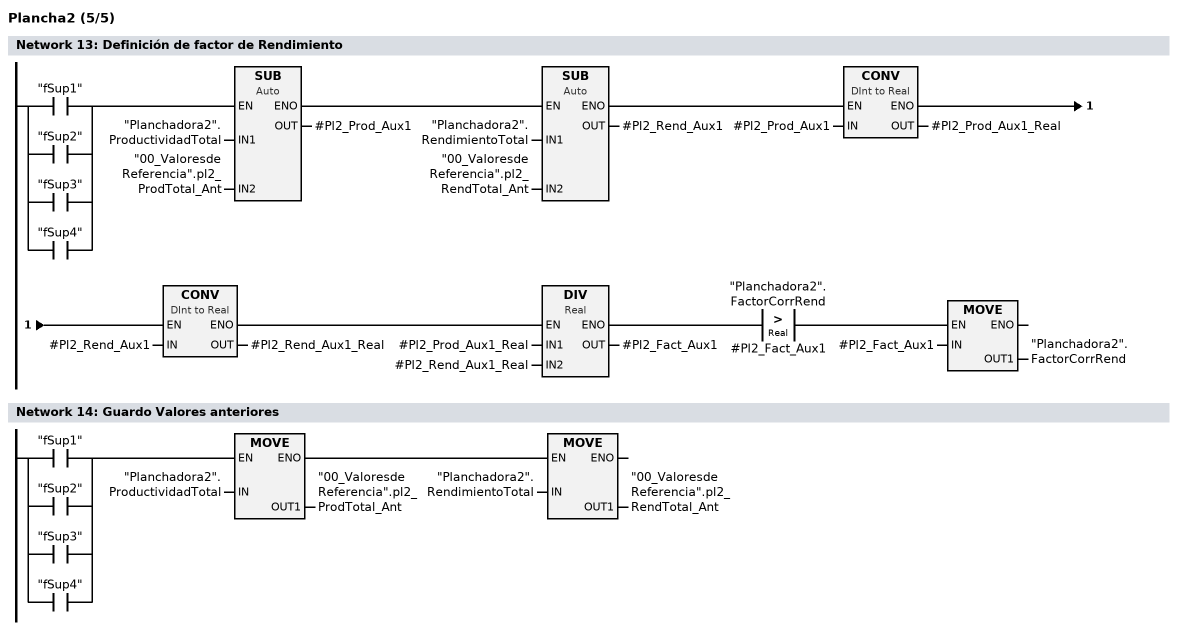
   RUNG wire#powerrail
      Contact( "fSup1" )
      wire#w1
      { S7_GenerateENO := "TRUE" } Sub(in1 := "Planchadora2".ProductividadTotal, in2 := "00_ValoresdeReferencia".pl2_ProdTotal_Ant, out => #Pl2_Prod_Aux1)
      { S7_GenerateENO := "TRUE" } Sub(in1 := "Planchadora2".RendimientoTotal, in2 := "00_ValoresdeReferencia".pl2_RendTotal_Ant, out => #Pl2_Rend_Aux1)
      { S7_Templates := "[SrcType := DInt, DestType := Real]"; S7_GenerateENO := "TRUE" } Convert(in := #Pl2_Prod_Aux1, out => #Pl2_Prod_Aux1_Real)
      { S7_Templates := "[SrcType := DInt, DestType := Real]"; S7_GenerateENO := "TRUE" } Convert(in := #Pl2_Rend_Aux1, out => #Pl2_Rend_Aux1_Real)
      { S7_Templates := "SrcType := Real"; S7_GenerateENO := "TRUE" } Div(in1 := #Pl2_Prod_Aux1_Real, in2 := #Pl2_Rend_Aux1_Real, out => #Pl2_Fact_Aux1)
      { S7_Templates := "SrcType := Real" } GT_Contact(in1 := "Planchadora2".FactorCorrRend, in2 := #Pl2_Fact_Aux1)
      { S7_GenerateENO := "TRUE" } Move(in := #Pl2_Fact_Aux1, out1 => "Planchadora2".FactorCorrRend)
   END_RUNG
   RUNG wire#powerrail
      Contact( "fSup2" )
   END_RUNG wire#w1
   RUNG wire#powerrail
      Contact( "fSup3" )
   END_RUNG wire#w1
   RUNG wire#powerrail
      Contact( "fSup4" )
   END_RUNG wire#w1
   // the same network as SCL:
   // ENO of a box is taken as its EN; it also drops when the box reports an error
   #_w1 := "fSup1" OR "fSup2" OR "fSup3" OR "fSup4";
   IF #_w1 THEN
       #Pl2_Prod_Aux1 := "Planchadora2".ProductividadTotal - "00_ValoresdeReferencia".pl2_ProdTotal_Ant;
       #Pl2_Rend_Aux1 := "Planchadora2".RendimientoTotal - "00_ValoresdeReferencia".pl2_RendTotal_Ant;
       #Pl2_Prod_Aux1_Real := DINT_TO_REAL(#Pl2_Prod_Aux1);
       #Pl2_Rend_Aux1_Real := DINT_TO_REAL(#Pl2_Rend_Aux1);
       #Pl2_Fact_Aux1 := #Pl2_Prod_Aux1_Real / #Pl2_Rend_Aux1_Real;
   END_IF;
   IF #_w1 AND ("Planchadora2".FactorCorrRend > #Pl2_Fact_Aux1) THEN
       "Planchadora2".FactorCorrRend := #Pl2_Fact_Aux1;
   END_IF;
END_REGION

REGION Network 14: Guardo Valores anteriores
   RUNG wire#powerrail
      Contact( "fSup1" )
      wire#w1
      { S7_GenerateENO := "TRUE" } Move(in := "Planchadora2".ProductividadTotal, out1 => "00_ValoresdeReferencia".pl2_ProdTotal_Ant)
      { S7_GenerateENO := "TRUE" } Move(in := "Planchadora2".RendimientoTotal, out1 => "00_ValoresdeReferencia".pl2_RendTotal_Ant)
   END_RUNG
   RUNG wire#powerrail
      Contact( "fSup2" )
   END_RUNG wire#w1
   RUNG wire#powerrail
      Contact( "fSup3" )
   END_RUNG wire#w1
   RUNG wire#powerrail
      Contact( "fSup4" )
   END_RUNG wire#w1
   // the same network as SCL:
   // ENO of a box is taken as its EN; it also drops when the box reports an error
   IF "fSup1" OR "fSup2" OR "fSup3" OR "fSup4" THEN
       "00_ValoresdeReferencia".pl2_ProdTotal_Ant := "Planchadora2".ProductividadTotal;
       "00_ValoresdeReferencia".pl2_RendTotal_Ant := "Planchadora2".RendimientoTotal;
   END_IF;
END_REGION
END_FUNCTION

FUNCTION "FC_Alarmas" : Void   // FC4, LAD
{ S7_Optimized_Access := 'FALSE' }
VERSION : 0.1
   VAR_TEMP
      tmp_Reconocimiento_1 : Word;
      tmp_Reconocimiento_2 : Word;
      tmp_Reconocidas_1 : Word;
      tmp_Reconocidas_2 : Word;
   END_VAR
BEGIN

REGION Network 1: PLANCHADORA 1
END_REGION

REGION Network 2: Falla Sensor Izquierda
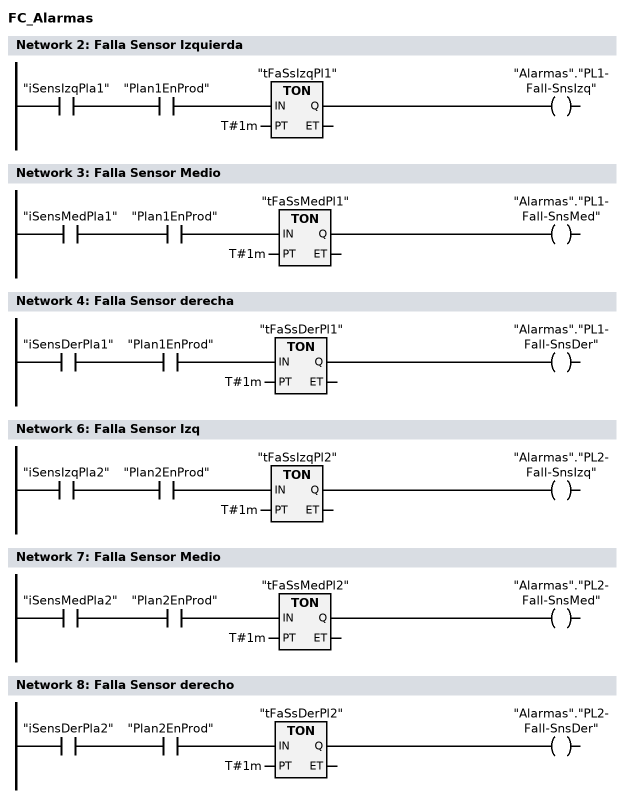
   "tFaSsIzqPl1".TON(IN := "iSensIzqPla1" AND "Plan1EnProd", PT := T#1m);
   "Alarmas"."PL1-Fall-SnsIzq" := "tFaSsIzqPl1".Q;
END_REGION

REGION Network 3: Falla Sensor Medio
   "tFaSsMedPl1".TON(IN := "iSensMedPla1" AND "Plan1EnProd", PT := T#1m);
   "Alarmas"."PL1-Fall-SnsMed" := "tFaSsMedPl1".Q;
END_REGION

REGION Network 4: Falla Sensor derecha
   "tFaSsDerPl1".TON(IN := "iSensDerPla1" AND "Plan1EnProd", PT := T#1m);
   "Alarmas"."PL1-Fall-SnsDer" := "tFaSsDerPl1".Q;
END_REGION

REGION Network 5: PLANCHADORA 2
END_REGION

REGION Network 6: Falla Sensor Izq
   "tFaSsIzqPl2".TON(IN := "iSensIzqPla2" AND "Plan2EnProd", PT := T#1m);
   "Alarmas"."PL2-Fall-SnsIzq" := "tFaSsIzqPl2".Q;
END_REGION

REGION Network 7: Falla Sensor Medio
   "tFaSsMedPl2".TON(IN := "iSensMedPla2" AND "Plan2EnProd", PT := T#1m);
   "Alarmas"."PL2-Fall-SnsMed" := "tFaSsMedPl2".Q;
END_REGION

REGION Network 8: Falla Sensor derecho
   "tFaSsDerPl2".TON(IN := "iSensDerPla2" AND "Plan2EnProd", PT := T#1m);
   "Alarmas"."PL2-Fall-SnsDer" := "tFaSsDerPl2".Q;
END_REGION
END_FUNCTION

FUNCTION "Simulacion" : Void   // FC5, LAD
{ S7_Optimized_Access := 'TRUE' }
VERSION : 0.1
BEGIN

REGION Network 1: Sensores Plancha 1
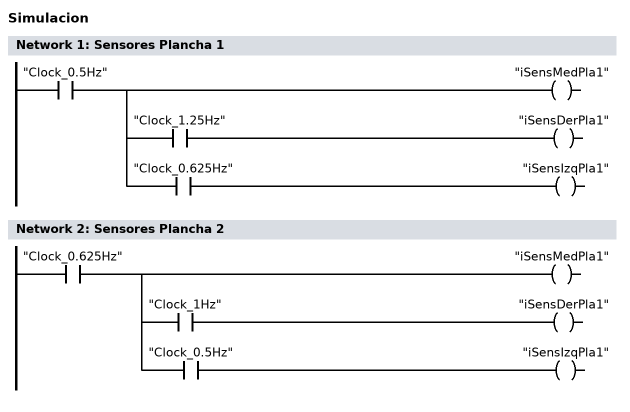
   RUNG wire#powerrail
      Contact( "Clock_0.5Hz" )
      wire#w1
      Coil( "iSensMedPla1" )
   END_RUNG
   RUNG wire#w1
      Contact( "Clock_1.25Hz" )
      Coil( "iSensDerPla1" )
   END_RUNG
   RUNG wire#w1
      Contact( "Clock_0.625Hz" )
      Coil( "iSensIzqPla1" )
   END_RUNG
   // the same network as SCL:
   "iSensMedPla1" := "Clock_0.5Hz";
   "iSensDerPla1" := "Clock_0.5Hz" AND "Clock_1.25Hz";
   "iSensIzqPla1" := "Clock_0.5Hz" AND "Clock_0.625Hz";
END_REGION

REGION Network 2: Sensores Plancha 2
   RUNG wire#powerrail
      Contact( "Clock_0.625Hz" )
      wire#w1
      Coil( "iSensMedPla1" )
   END_RUNG
   RUNG wire#w1
      Contact( "Clock_1Hz" )
      Coil( "iSensDerPla1" )
   END_RUNG
   RUNG wire#w1
      Contact( "Clock_0.5Hz" )
      Coil( "iSensIzqPla1" )
   END_RUNG
   // the same network as SCL:
   "iSensMedPla1" := "Clock_0.625Hz";
   "iSensDerPla1" := "Clock_0.625Hz" AND "Clock_1Hz";
   "iSensIzqPla1" := "Clock_0.625Hz" AND "Clock_0.5Hz";
END_REGION
END_FUNCTION

ORGANIZATION_BLOCK "Main"   // OB1, LAD, ProgramCycle
TITLE = "Main Program Sweep (Cycle)"
{ S7_Optimized_Access := 'TRUE' }
VERSION : 0.1
   VAR_TEMP
      Pl1_Prod_Aux1 : DInt;
      Pl1_Rend_Aux1 : DInt;
      Pl1_Fact_Aux1 : Real;
   END_VAR
   VAR_TEMP   // added for the SCL form of the ladder/FBD networks
      _w1 : Bool;
      _w2 : Bool;
   END_VAR
BEGIN

REGION Network 1: Flanco cada 15 minutos
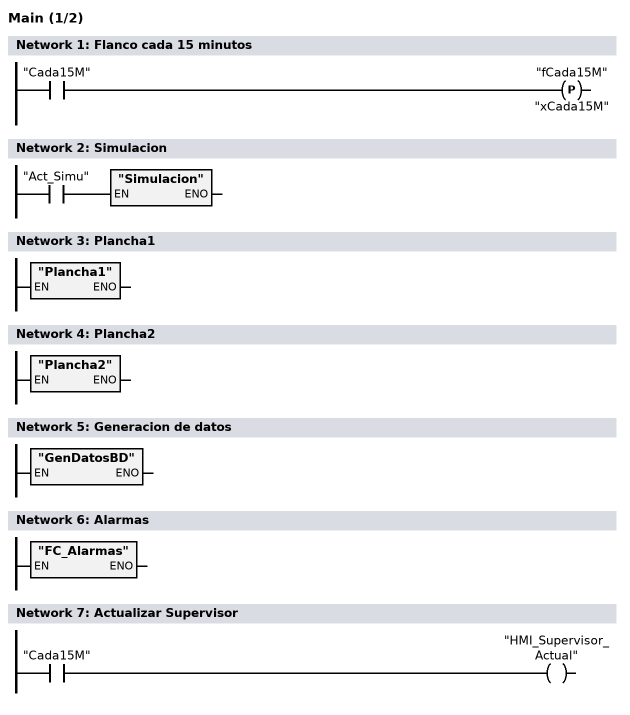
   "fCada15M" := "Cada15M" AND NOT "xCada15M";   // rising edge
   "xCada15M" := "Cada15M";
END_REGION

REGION Network 2: Simulacion
   RUNG wire#powerrail
      Contact( "Act_Simu" )
      "Simulacion"()
   END_RUNG
   // the same network as SCL:
   IF "Act_Simu" THEN "Simulacion"(); END_IF;
END_REGION

REGION Network 3: Plancha1
   RUNG wire#powerrail
      "Plancha1"()
   END_RUNG
   // the same network as SCL:
   "Plancha1"();
END_REGION

REGION Network 4: Plancha2
   RUNG wire#powerrail
      "Plancha2"()
   END_RUNG
   // the same network as SCL:
   "Plancha2"();
END_REGION

REGION Network 5: Generacion de datos
   RUNG wire#powerrail
      "GenDatosBD"()
   END_RUNG
   // the same network as SCL:
   "GenDatosBD"();
END_REGION

REGION Network 6: Alarmas
   RUNG wire#powerrail
      "FC_Alarmas"()
   END_RUNG
   // the same network as SCL:
   "FC_Alarmas"();
END_REGION

REGION Network 7: Actualizar Supervisor
   RUNG wire#powerrail
      Contact( "Cada15M" )
      Coil( "HMI_Supervisor_Actual" )
   END_RUNG
   // the same network as SCL:
   "HMI_Supervisor_Actual" := "Cada15M";
END_REGION

REGION Network 8: Oscilador de 5 minutos
   // Para refresco de grafica principal en WinCC
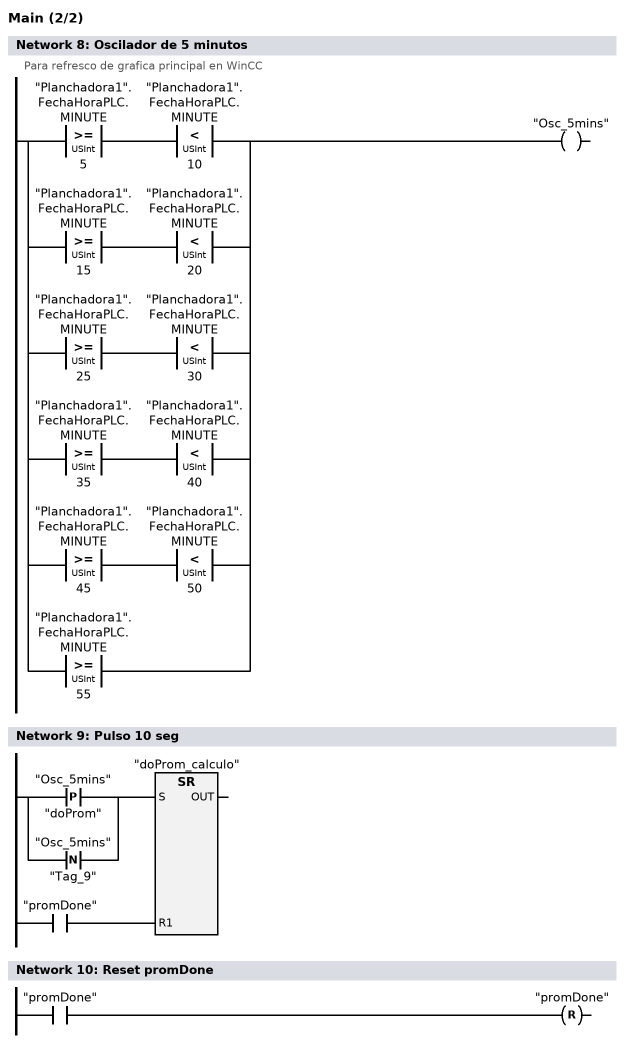
   RUNG wire#powerrail
      { S7_Templates := "SrcType := USInt" } GE_Contact(in1 := "Planchadora1".FechaHoraPLC.MINUTE, in2 := 5)
      { S7_Templates := "SrcType := USInt" } LT_Contact(in1 := "Planchadora1".FechaHoraPLC.MINUTE, in2 := 10)
      wire#w1
      Coil( "Osc_5mins" )
   END_RUNG
   RUNG wire#powerrail
      { S7_Templates := "SrcType := USInt" } GE_Contact(in1 := "Planchadora1".FechaHoraPLC.MINUTE, in2 := 15)
      { S7_Templates := "SrcType := USInt" } LT_Contact(in1 := "Planchadora1".FechaHoraPLC.MINUTE, in2 := 20)
   END_RUNG wire#w1
   RUNG wire#powerrail
      { S7_Templates := "SrcType := USInt" } GE_Contact(in1 := "Planchadora1".FechaHoraPLC.MINUTE, in2 := 25)
      { S7_Templates := "SrcType := USInt" } LT_Contact(in1 := "Planchadora1".FechaHoraPLC.MINUTE, in2 := 30)
   END_RUNG wire#w1
   RUNG wire#powerrail
      { S7_Templates := "SrcType := USInt" } GE_Contact(in1 := "Planchadora1".FechaHoraPLC.MINUTE, in2 := 35)
      { S7_Templates := "SrcType := USInt" } LT_Contact(in1 := "Planchadora1".FechaHoraPLC.MINUTE, in2 := 40)
   END_RUNG wire#w1
   RUNG wire#powerrail
      { S7_Templates := "SrcType := USInt" } GE_Contact(in1 := "Planchadora1".FechaHoraPLC.MINUTE, in2 := 45)
      { S7_Templates := "SrcType := USInt" } LT_Contact(in1 := "Planchadora1".FechaHoraPLC.MINUTE, in2 := 50)
   END_RUNG wire#w1
   RUNG wire#powerrail
      { S7_Templates := "SrcType := USInt" } GE_Contact(in1 := "Planchadora1".FechaHoraPLC.MINUTE, in2 := 55)
   END_RUNG wire#w1
   // the same network as SCL:
   "Osc_5mins" := (("Planchadora1".FechaHoraPLC.MINUTE >= 5) AND ("Planchadora1".FechaHoraPLC.MINUTE < 10)) OR (("Planchadora1".FechaHoraPLC.MINUTE >= 15) AND ("Planchadora1".FechaHoraPLC.MINUTE < 20)) OR (("Planchadora1".FechaHoraPLC.MINUTE >= 25) AND ("Planchadora1".FechaHoraPLC.MINUTE < 30)) OR (("Planchadora1".FechaHoraPLC.MINUTE >= 35) AND ("Planchadora1".FechaHoraPLC.MINUTE < 40)) OR (("Planchadora1".FechaHoraPLC.MINUTE >= 45) AND ("Planchadora1".FechaHoraPLC.MINUTE < 50)) OR ("Planchadora1".FechaHoraPLC.MINUTE >= 55);
END_REGION

REGION Network 9: Pulso 10 seg
   RUNG wire#powerrail
      P_Contact(operand := "Osc_5mins", bit := "doProm")
      wire#w1
      S_SR(operand := "doProm_calculo", r1 := wire#w2)
   END_RUNG
   RUNG wire#powerrail
      N_Contact(operand := "Osc_5mins", bit := "Tag_9")
   END_RUNG wire#w1
   RUNG wire#powerrail
      Contact( "promDone" )
   END_RUNG wire#w2
   // the same network as SCL:
   #_w1 := "Osc_5mins" AND NOT "doProm";   // rising edge of "Osc_5mins"
   "doProm" := "Osc_5mins";
   #_w2 := NOT "Osc_5mins" AND "Tag_9";   // falling edge of "Osc_5mins"
   "Tag_9" := "Osc_5mins";
   IF #_w1 OR #_w2 THEN
       "doProm_calculo" := TRUE;   // SR flip-flop
   END_IF;
   IF "promDone" THEN "doProm_calculo" := FALSE; END_IF;
END_REGION

REGION Network 10: Reset promDone
   RUNG wire#powerrail
      Contact( "promDone" )
      R_Coil( "promDone" )
   END_RUNG
   // the same network as SCL:
   IF "promDone" THEN "promDone" := FALSE; END_IF;
END_REGION
END_ORGANIZATION_BLOCK

(* ===== HMI "HMI_RT_1" =====
system functions are stored by id; their names below are inferred from use
connection "Lav_Broun_3": COM3, MODBUS_RTU
connection "HMI_Conexión_1": ETHERNET, S7_1200_OMS
connection "Lav_Broun_2": COM3, MODBUS_RTU
connection "Lav_Broun_1": COM3, MODBUS_RTU
connection "Lav_Broun_4": COM3, MODBUS_RTU

HMI tags "Tabla de variables estándar"
   "MaqEnProd" : Bool = PLC Plan1EnProd AT %M2.2, 1 s
   "Cada15M" : Bool = PLC Cada15M AT %M3.4, 1 s
      on ChangeValue: "S03_Write_data_record_into_a_table"()
   "AnoPLC" : UInt = PLC Planchadora1.FechaHoraPLC.YEAR AT %DB1.DBW0, 1 s
      on ChangeValue: "S07_InformeDiario_Planchas"(N)
   "MesPLC" : USInt = PLC Planchadora1.FechaHoraPLC.MONTH AT %DB1.DBW0, 1 s
   "DiaPLC" : USInt = PLC Planchadora1.FechaHoraPLC.DAY AT %DB1.DBW0, 1 s
   "tmp_prueba_0" : WString[100], internal
   "tmp_prueba_1" : WString[100], internal
   "tmp_prueba_2" : WString[100], internal
   "tmp_prueba_3" : WString[100], internal
   "tmp_prueba_4" : WString[100], internal
   "tmp_prueba_5" : DateTime, internal
   "Inf_FechaInforme_WeekDay" : Int, internal
   "Inf_FechaInforme" : DateTime, internal
   "Planchadora2_FactorCorrRend" : Real = PLC Planchadora2.FactorCorrRend, 1 s
   "iSensIzqPla1" : Bool = PLC iSensIzqPla1 AT %I0.0, 1 s
   "BCDtoInt" : WString[10] AT %DB1.DBX0.0
   "BCDtoInt_Entrada" : DateTime, internal
   "bitmask" : Int, internal
   "Indices_objetivo_100" : Real = PLC Indices.objetivo_100, 1 s
   "Indices_horasTurno" : Time_Of_Day = PLC Indices.horasTurno, 1 s
   "Indices_objetivo" : Time_Of_Day = PLC Indices.objetivo, 1 s
   "Indices_avance" : Time_Of_Day = PLC Indices.avance, 1 s
   "Indices_avance_100" : Real = PLC Indices.avance_100, 1 s
   "Indices_real" : Time_Of_Day = PLC Indices.avance_real, 1 s
   "Indices_avance_real_100" : Real = PLC Indices.avance_real_100, 1 s
   "Osc_5mins" : Bool = PLC Osc_5mins AT %M100.0, 5 s
   "Ala-Disp-W0" : Word AT %DB9.DBW0, 1 s
   "Ala-Disp-W1" : Word AT %DB9.DBW1, 1 s
   "Indices_avance_100_tReal" : Real = PLC Indices.avance_100, 1 s
   "Indices_objetivo_100_tReal" : Real = PLC Indices.objetivo_100, 1 s
   "Indices_avance_real_100_tReal" : Real = PLC Indices.avance_real_100, 1 s
   "Planchadora1_Tiempo" : DInt = PLC Planchadora1.Tiempo, 1 s
   "Planchadora2_Productividad" : DInt = PLC Planchadora2.Productividad, 1 s
   "Planchadora2_Rendimiento" : DInt = PLC Planchadora2.Rendimiento, 1 s
   "Planchadora2_Tiempo" : DInt = PLC Planchadora2.Tiempo, 1 s
   "Alarmas_PL1-Fall-SnsIzq" : Bool = PLC Alarmas.PL1-Fall-SnsIzq AT %DB9.DBX0.0, 1 s
      on ChangeValue: "SA5_email_SnsPlancha"(1, 'Norte')
   "Alarmas_PL1-Fall-SnsMed" : Bool = PLC Alarmas.PL1-Fall-SnsMed AT %DB9.DBX0.1, 1 s
      on ChangeValue: "SA5_email_SnsPlancha"(1, 'Centro')
   "Alarmas_PL1-Fall-SnsDer" : Bool = PLC Alarmas.PL1-Fall-SnsDer AT %DB9.DBX0.2, 1 s
      on ChangeValue: "SA5_email_SnsPlancha"(1, 'Sur')
   "Alarmas_PL2-Fall-SnsIzq" : Bool = PLC Alarmas.PL2-Fall-SnsIzq AT %DB9.DBX0.3, 1 s
      on ChangeValue: "SA5_email_SnsPlancha"(2, 'Norte')
   "Alarmas_PL2-Fall-SnsMed" : Bool = PLC Alarmas.PL2-Fall-SnsMed AT %DB9.DBX0.4, 1 s
      on ChangeValue: "SA5_email_SnsPlancha"(2, 'Centro')
   "Alarmas_PL2-Fall-SnsDer" : Bool = PLC Alarmas.PL2-Fall-SnsDer AT %DB9.DBX0.5, 1 s
      on ChangeValue: "SA5_email_SnsPlancha"(2, 'Sur')

HMI tags "ListaClientes"
   "ID_1" : Int, internal
   "ID_2" : Int, internal
   "ID_3" : Int, internal
   "ID_4" : Int, internal
   "ID_5" : Int, internal
   "Name_1" : WString[64], internal
   "Name_2" : WString[64], internal
   "Name_3" : WString[64], internal
   "Name_4" : WString[64], internal
   "Name_5" : WString[64], internal
   "ID_Cambiar" : Int, internal
   "Name_Cambiar" : WString[64], internal
   "ID_Nuevo" : Int, internal
   "Name_Nuevo" : WString[64], internal
   "Cli_ID" : Int AT %DB1.DBW0
   "Cli_Name" : WString[254] AT %DB1.DBX0.0

